C07289=1074.285,247.600,415.583,174.405,27.712,154.898
C07290=1074.292,247.848,415.555,174.407,27.716,154.899
C07291=1074.297,248.097,415.528,174.409,27.720,154.899
C07292=1074.302,248.345,415.500,174.412,27.724,154.900
C07293=1074.309,248.594,415.472,174.415,27.728,154.900
C07294=1074.318,249.000,415.427,174.419,27.734,154.901
C07295=1074.327,249.406,415.383,174.423,27.740,154.902
C07296=1074.336,249.812,415.337,174.427,27.746,154.903
C07297=1074.345,250.218,415.292,174.430,27.753,154.904
C07298=1074.351,250.466,415.265,174.433,27.757,154.905
C07299=1074.357,250.714,415.236,174.435,27.761,154.905
C07300=1074.362,250.963,415.209,174.437,27.765,154.906
C07301=1074.368,251.211,415.182,174.440,27.768,154.907
C07302=1074.374,251.459,415.153,174.442,27.772,154.907
C07303=1074.379,251.708,415.126,174.445,27.777,154.908
C07304=1074.386,251.957,415.098,174.448,27.780,154.908
C07305=1074.391,252.205,415.070,174.450,27.784,154.909
C07306=1074.397,252.453,415.042,174.452,27.788,154.910
C07307=1074.404,252.701,415.015,174.455,27.792,154.910
C07308=1074.409,252.950,414.988,174.457,27.796,154.911
C07309=1074.414,253.199,414.959,174.459,27.799,154.911
C07310=1074.421,253.446,414.932,174.462,27.803,154.912
C07311=1074.427,253.695,414.904,174.465,27.807,154.913
C07312=1074.432,253.943,414.876,174.467,27.811,154.913
C07313=1074.438,254.192,414.847,174.470,27.815,154.914
C07314=1074.444,254.440,414.821,174.472,27.819,154.914
C07315=1074.450,254.689,414.792,174.474,27.822,154.915
C07316=1074.455,254.937,414.764,174.476,27.826,154.916
C07317=1074.462,255.185,414.737,174.479,27.830,154.916
C07318=1074.467,255.433,414.709,174.482,27.834,154.917
C07319=1074.473,255.682,414.680,174.484,27.838,154.917
C07320=1074.478,255.930,414.652,174.487,27.842,154.918
C07321=1074.485,256.179,414.625,174.489,27.846,154.919
C07322=1074.491,256.427,414.596,174.492,27.849,154.919
C07323=1074.496,256.676,414.568,174.494,27.853,154.920
C07324=1074.502,256.924,414.540,174.497,27.857,154.920
C07325=1074.508,257.172,414.513,174.499,27.861,154.921
C07326=1074.514,257.421,414.484,174.502,27.865,154.922
C07327=1074.519,257.669,414.456,174.504,27.868,154.922
C07328=1074.525,257.918,414.428,174.507,27.872,154.923
C07329=1074.531,258.166,414.400,174.509,27.876,154.923
C07330=1074.537,258.414,414.372,174.512,27.880,154.924
C07331=1074.544,258.662,414.343,174.515,27.884,154.924
C07332=1074.550,258.911,414.315,174.517,27.888,154.925
C07333=1074.555,259.159,414.287,174.519,27.892,154.926
C07334=1074.562,259.407,414.259,174.522,27.895,154.926
C07335=1074.567,259.655,414.231,174.524,27.899,154.927
C07336=1074.573,259.904,414.203,174.527,27.903,154.927
C07337=1074.579,260.152,414.174,174.530,27.907,154.928
C07338=1074.584,260.400,414.146,174.532,27.910,154.929
C07339=1074.590,260.649,414.118,174.534,27.914,154.929
C07340=1074.597,260.898,414.090,174.537,27.918,154.930
C07341=1074.603,261.146,414.062,174.540,27.922,154.930
C07342=1074.609,261.394,414.033,174.542,27.926,154.931
C07343=1074.615,261.643,414.005,174.545,27.930,154.932
C07344=1074.621,261.891,413.976,174.547,27.934,154.932
C07345=1074.626,262.139,413.948,174.549,27.937,154.933
C07346=1074.636,262.543,413.902,174.554,27.944,154.934
C07347=1074.646,262.946,413.856,174.558,27.950,154.935
C07348=1074.656,263.349,413.810,174.562,27.956,154.936
C07349=1074.666,263.753,413.764,174.566,27.962,154.937
C07350=1074.672,264.002,413.735,174.569,27.966,154.937
C07351=1074.677,264.249,413.707,174.572,27.970,154.938
C07352=1074.683,264.498,413.678,174.574,27.974,154.938
C07353=1074.689,264.746,413.649,174.576,27.978,154.939
C07354=1074.695,264.994,413.621,174.579,27.981,154.939
C07355=1074.700,265.242,413.592,174.582,27.985,154.940
C07356=1074.706,265.491,413.563,174.584,27.989,154.941
C07357=1074.713,265.739,413.534,174.587,27.993,154.941
C07358=1074.718,265.987,413.506,174.589,27.997,154.942
C07359=1074.724,266.235,413.477,174.592,28.001,154.943
C07360=1074.730,266.484,413.449,174.595,28.005,154.943
C07361=1074.735,266.732,413.420,174.597,28.009,154.944
C07362=1074.741,266.980,413.391,174.600,28.013,154.944
C07363=1074.747,267.229,413.362,174.603,28.017,154.945
C07364=1074.753,267.477,413.333,174.605,28.020,154.946
C07365=1074.759,267.726,413.305,174.608,28.024,154.946
C07366=1074.765,267.973,413.276,174.610,28.028,154.947
C07367=1074.771,268.222,413.247,174.613,28.032,154.947
C07368=1074.776,268.470,413.218,174.616,28.036,154.948
C07369=1074.783,268.718,413.189,174.618,28.040,154.949
C07370=1074.789,268.967,413.160,174.620,28.044,154.949
C07371=1074.795,269.214,413.131,174.624,28.048,154.950
C07372=1074.800,269.463,413.103,174.626,28.052,154.950
C07373=1074.806,269.711,413.074,174.628,28.056,154.951
C07374=1074.812,269.959,413.044,174.631,28.059,154.952
C07375=1074.818,270.208,413.015,174.634,28.063,154.952
C07376=1074.823,270.456,412.987,174.636,28.067,154.953
C07377=1074.829,270.704,412.958,174.639,28.071,154.953
C07378=1074.835,270.952,412.928,174.641,28.075,154.954
C07379=1074.841,271.201,412.899,174.644,28.079,154.955
C07380=1074.847,271.449,412.870,174.647,28.083,154.955
C07381=1074.853,271.698,412.841,174.649,28.087,154.956
C07382=1074.859,271.946,412.812,174.651,28.091,154.957
C07383=1074.865,272.193,412.784,174.655,28.095,154.957
C07384=1074.870,272.442,412.754,174.657,28.099,154.958
C07385=1074.876,272.690,412.725,174.660,28.102,154.958
C07386=1074.883,272.938,412.696,174.663,28.107,154.959
C07387=1074.888,273.186,412.666,174.665,28.110,154.960
C07388=1074.894,273.435,412.637,174.668,28.114,154.960
C07389=1074.900,273.683,412.607,174.670,28.118,154.961
C07390=1074.906,273.931,412.578,174.673,28.122,154.961
C07391=1074.912,274.180,412.549,174.676,28.126,154.962
C07392=1074.918,274.428,412.520,174.678,28.130,154.963
C07393=1074.923,274.675,412.490,174.681,28.134,154.963
C07394=1074.929,274.924,412.461,174.684,28.138,154.964
C07395=1074.934,275.172,412.432,174.686,28.142,154.965
C07396=1074.941,275.420,412.403,174.688,28.146,154.965
C07397=1074.946,275.669,412.373,174.692,28.150,154.966
C07398=1074.956,276.076,412.325,174.696,28.156,154.967
C07399=1074.966,276.482,412.277,174.700,28.163,154.968
C07400=1074.976,276.888,412.229,174.704,28.169,154.969
C07401=1074.985,277.294,412.180,174.708,28.176,154.970
C07402=1074.991,277.543,412.151,174.712,28.180,154.971
C07403=1074.996,277.791,412.121,174.714,28.183,154.971
C07404=1075.003,278.039,412.092,174.716,28.187,154.972
C07405=1075.008,278.288,412.062,174.720,28.192,154.972
C07406=1075.014,278.535,412.032,174.722,28.196,154.973
C07407=1075.020,278.783,412.003,174.724,28.200,154.974
C07408=1075.026,279.032,411.973,174.728,28.203,154.974
C07409=1075.032,279.279,411.944,174.730,28.207,154.975
C07410=1075.038,279.528,411.914,174.733,28.211,154.975
C07411=1075.043,279.776,411.884,174.736,28.215,154.976
C07412=1075.050,280.025,411.854,174.738,28.219,154.977
C07413=1075.056,280.273,411.825,174.741,28.223,154.977
C07414=1075.061,280.521,411.795,174.744,28.227,154.978
C07415=1075.068,280.769,411.765,174.746,28.231,154.979
C07416=1075.074,281.017,411.736,174.749,28.235,154.979
C07417=1075.079,281.266,411.706,174.752,28.239,154.980
C07418=1075.085,281.514,411.676,174.754,28.243,154.980
C07419=1075.091,281.762,411.647,174.758,28.247,154.981
C07420=1075.097,282.010,411.616,174.760,28.251,154.982
C07421=1075.102,282.258,411.587,174.762,28.255,154.982
C07422=1075.108,282.506,411.556,174.766,28.260,154.983
C07423=1075.114,282.754,411.527,174.768,28.263,154.984
C07424=1075.120,283.002,411.496,174.770,28.267,154.984
C07425=1075.126,283.250,411.467,174.774,28.272,154.985
C07426=1075.132,283.498,411.437,174.776,28.275,154.986
C07427=1075.137,283.746,411.406,174.779,28.279,154.986
C07428=1075.143,283.994,411.377,174.782,28.283,154.987
C07429=1075.149,284.243,411.346,174.784,28.287,154.987
C07430=1075.155,284.491,411.317,174.788,28.291,154.988
C07431=1075.161,284.739,411.286,174.790,28.295,154.989
C07432=1075.167,284.987,411.256,174.792,28.299,154.989
C07433=1075.173,285.235,411.227,174.796,28.304,154.990
C07434=1075.179,285.483,411.196,174.798,28.308,154.991
C07435=1075.184,285.731,411.166,174.800,28.311,154.991
C07436=1075.191,285.980,411.136,174.804,28.316,154.992
C07437=1075.196,286.228,411.106,174.806,28.320,154.993
C07438=1075.202,286.476,411.075,174.809,28.324,154.993
C07439=1075.208,286.723,411.045,174.812,28.328,154.994
C07440=1075.213,286.972,411.015,174.814,28.332,154.995
C07441=1075.220,287.219,410.986,174.817,28.336,154.995
C07442=1075.226,287.468,410.955,174.820,28.339,154.996
C07443=1075.232,287.716,410.925,174.823,28.344,154.996
C07444=1075.238,287.964,410.895,174.826,28.348,154.997
C07445=1075.244,288.212,410.865,174.828,28.352,154.998
C07446=1075.250,288.460,410.834,174.831,28.356,154.998
C07447=1075.256,288.708,410.804,174.834,28.360,154.999
C07448=1075.262,288.956,410.773,174.837,28.364,155.000
C07449=1075.267,289.204,410.743,174.839,28.368,155.000
C07450=1075.277,289.621,410.692,174.844,28.375,155.001
C07451=1075.288,290.038,410.641,174.849,28.381,155.002
C07452=1075.297,290.454,410.590,174.853,28.389,155.004
C07453=1075.307,290.870,410.538,174.858,28.395,155.005
C07454=1075.313,291.118,410.507,174.861,28.400,155.005
C07455=1075.319,291.367,410.477,174.864,28.404,155.006
C07456=1075.325,291.615,410.446,174.866,28.408,155.007
C07457=1075.331,291.862,410.416,174.869,28.412,155.007
C07458=1075.337,292.110,410.386,174.872,28.416,155.008
C07459=1075.343,292.359,410.355,174.875,28.420,155.009
C07460=1075.348,292.607,410.324,174.878,28.424,155.009
C07461=1075.354,292.855,410.294,174.881,28.428,155.010
C07462=1075.360,293.103,410.263,174.883,28.432,155.011
C07463=1075.366,293.350,410.232,174.887,28.437,155.011
C07464=1075.372,293.598,410.202,174.889,28.441,155.012
C07465=1075.378,293.847,410.170,174.891,28.445,155.013
C07466=1075.384,294.095,410.140,174.895,28.449,155.013
C07467=1075.390,294.343,410.110,174.897,28.453,155.014
C07468=1075.396,294.591,410.078,174.900,28.457,155.015
C07469=1075.402,294.839,410.048,174.903,28.461,155.015
C07470=1075.407,295.087,410.017,174.906,28.465,155.016
C07471=1075.414,295.335,409.986,174.909,28.469,155.016
C07472=1075.420,295.582,409.955,174.912,28.474,155.017
C07473=1075.426,295.831,409.924,174.914,28.478,155.018
C07474=1075.431,296.079,409.893,174.918,28.482,155.019
C07475=1075.437,296.326,409.862,174.920,28.486,155.019
C07476=1075.444,296.575,409.832,174.923,28.490,155.020
C07477=1075.449,296.823,409.801,174.926,28.494,155.021
C07478=1075.455,297.070,409.770,174.929,28.498,155.021
C07479=1075.461,297.319,409.739,174.931,28.502,155.022
C07480=1075.466,297.567,409.708,174.935,28.507,155.023
C07481=1075.473,297.815,409.676,174.937,28.511,155.023
C07482=1075.478,298.063,409.646,174.940,28.515,155.024
C07483=1075.484,298.310,409.614,174.943,28.519,155.025
C07484=1075.490,298.559,409.583,174.946,28.523,155.025
C07485=1075.495,298.806,409.551,174.948,28.528,155.026
C07486=1075.501,299.054,409.521,174.952,28.532,155.027
C07487=1075.507,299.302,409.489,174.954,28.536,155.027
C07488=1075.513,299.550,409.458,174.957,28.541,155.028
C07489=1075.519,299.798,409.427,174.960,28.545,155.029
C07490=1075.524,300.046,409.395,174.963,28.549,155.029
C07491=1075.530,300.294,409.365,174.966,28.553,155.030
C07492=1075.536,300.542,409.333,174.969,28.558,155.031
C07493=1075.542,300.789,409.302,174.971,28.562,155.032
C07494=1075.548,301.038,409.270,174.975,28.566,155.032
C07495=1075.553,301.285,409.239,174.977,28.570,155.033
C07496=1075.560,301.533,409.207,174.980,28.575,155.034
C07497=1075.565,301.782,409.176,174.983,28.579,155.034
C07498=1075.572,302.029,409.145,174.986,28.583,155.035
C07499=1075.577,302.277,409.113,174.988,28.587,155.036
C07500=1075.582,302.525,409.082,174.992,28.592,155.036
C07501=1075.589,302.773,409.051,174.994,28.596,155.037
C07502=1075.594,302.988,409.023,174.996,28.600,155.038
C07503=1075.599,303.204,408.995,174.999,28.603,155.038
C07504=1075.605,303.420,408.968,175.002,28.607,155.039
C07505=1075.609,303.635,408.941,175.005,28.611,155.040
C07506=1075.615,303.851,408.913,175.007,28.614,155.040
C07507=1075.620,304.066,408.886,175.010,28.618,155.041
C07508=1075.625,304.282,408.859,175.012,28.622,155.041
C07509=1075.630,304.498,408.832,175.015,28.626,155.042
C07510=1075.636,304.746,408.800,175.018,28.630,155.043
C07511=1075.642,304.994,408.768,175.020,28.634,155.043
C07512=1075.648,305.241,408.737,175.024,28.638,155.044
C07513=1075.654,305.489,408.705,175.026,28.643,155.045
C07514=1075.659,305.737,408.673,175.029,28.647,155.046
C07515=1075.666,305.985,408.641,175.032,28.651,155.046
C07516=1075.671,306.232,408.610,175.035,28.656,155.047
C07517=1075.677,306.481,408.578,175.038,28.660,155.048
C07518=1075.684,306.728,408.546,175.041,28.664,155.048
C07519=1075.689,306.976,408.515,175.044,28.668,155.049
C07520=1075.695,307.224,408.483,175.046,28.673,155.050
C07521=1075.701,307.472,408.451,175.050,28.677,155.050
C07522=1075.707,307.720,408.420,175.052,28.681,155.051
C07523=1075.713,307.968,408.388,175.056,28.686,155.052
C07524=1075.719,308.216,408.356,175.059,28.690,155.053
C07525=1075.725,308.464,408.324,175.061,28.694,155.053
C07526=1075.731,308.711,408.292,175.065,28.699,155.054
C07527=1075.738,308.959,408.260,175.067,28.703,155.055
C07528=1075.743,309.207,408.228,175.070,28.707,155.055
C07529=1075.749,309.455,408.196,175.074,28.712,155.056
C07530=1075.756,309.703,408.165,175.076,28.716,155.057
C07531=1075.762,309.951,408.133,175.079,28.720,155.058
C07532=1075.767,310.198,408.101,175.083,28.725,155.058
C07533=1075.773,310.446,408.068,175.085,28.729,155.059
C07534=1075.779,310.694,408.036,175.088,28.733,155.060
C07535=1075.786,310.942,408.005,175.091,28.737,155.060
C07536=1075.792,311.190,407.973,175.094,28.742,155.061
C07537=1075.798,311.437,407.940,175.098,28.746,155.062
C07538=1075.804,311.685,407.908,175.100,28.751,155.063
C07539=1075.810,311.934,407.876,175.103,28.755,155.063
C07540=1075.816,312.181,407.843,175.107,28.759,155.064
C07541=1075.823,312.429,407.812,175.109,28.763,155.065
C07542=1075.828,312.677,407.780,175.112,28.768,155.065
C07543=1075.835,312.924,407.748,175.115,28.772,155.066
C07544=1075.841,313.172,407.716,175.118,28.776,155.067
C07545=1075.847,313.420,407.683,175.121,28.781,155.068
C07546=1075.853,313.668,407.651,175.124,28.785,155.068
C07547=1075.859,313.916,407.619,175.127,28.790,155.069
C07548=1075.866,314.164,407.587,175.131,28.794,155.070
C07549=1075.871,314.411,407.555,175.133,28.798,155.070
C07550=1075.877,314.659,407.522,175.136,28.803,155.071
C07551=1075.883,314.907,407.490,175.140,28.807,155.072
C07552=1075.889,315.155,407.457,175.142,28.811,155.073
C07553=1075.895,315.403,407.425,175.145,28.816,155.073
C07554=1075.901,315.650,407.393,175.149,28.821,155.074
C07555=1075.906,315.898,407.359,175.151,28.825,155.075
C07556=1075.912,316.146,407.327,175.154,28.830,155.076
C07557=1075.919,316.394,407.294,175.157,28.834,155.077
C07558=1075.924,316.611,407.266,175.160,28.838,155.077
C07559=1075.928,316.828,407.237,175.163,28.842,155.078
C07560=1075.933,317.045,407.209,175.165,28.846,155.079
C07561=1075.938,317.262,407.180,175.168,28.850,155.079
C07562=1075.944,317.480,407.151,175.171,28.854,155.080
C07563=1075.949,317.697,407.123,175.173,28.858,155.081
C07564=1075.954,317.914,407.094,175.176,28.862,155.081
C07565=1075.959,318.131,407.065,175.178,28.866,155.082
C07566=1075.965,318.379,407.033,175.182,28.871,155.083
C07567=1075.972,318.627,407.000,175.185,28.876,155.083
C07568=1075.977,318.875,406.967,175.187,28.880,155.084
C07569=1075.983,319.123,406.934,175.191,28.885,155.085
C07570=1075.989,319.371,406.901,175.194,28.889,155.086
C07571=1075.995,319.618,406.868,175.196,28.894,155.087
C07572=1076.001,319.866,406.836,175.200,28.898,155.087
C07573=1076.007,320.114,406.803,175.203,28.903,155.088
C07574=1076.013,320.362,406.770,175.205,28.907,155.089
C07575=1076.019,320.609,406.738,175.209,28.912,155.090
C07576=1076.024,320.857,406.705,175.212,28.917,155.090
C07577=1076.030,321.104,406.672,175.214,28.921,155.091
C07578=1076.036,321.352,406.638,175.218,28.926,155.092
C07579=1076.042,321.600,406.606,175.221,28.930,155.093
C07580=1076.049,321.847,406.573,175.224,28.935,155.094
C07581=1076.055,322.096,406.539,175.227,28.939,155.094
C07582=1076.061,322.344,406.507,175.230,28.944,155.095
C07583=1076.067,322.591,406.473,175.233,28.949,155.096
C07584=1076.073,322.839,406.440,175.236,28.953,155.097
C07585=1076.078,323.087,406.407,175.239,28.958,155.097
C07586=1076.085,323.335,406.374,175.243,28.963,155.098
C07587=1076.091,323.582,406.342,175.246,28.967,155.099
C07588=1076.096,323.830,406.308,175.248,28.972,155.100
C07589=1076.103,324.078,406.276,175.252,28.976,155.101
C07590=1076.109,324.325,406.242,175.255,28.981,155.101
C07591=1076.115,324.573,406.209,175.258,28.986,155.102
C07592=1076.120,324.820,406.175,175.261,28.990,155.103
C07593=1076.127,325.069,406.142,175.264,28.995,155.104
C07594=1076.133,325.317,406.109,175.267,29.000,155.105
C07595=1076.139,325.564,406.076,175.271,29.004,155.105
C07596=1076.145,325.812,406.042,175.273,29.009,155.106
C07597=1076.151,326.059,406.009,175.276,29.013,155.107
C07598=1076.157,326.307,405.976,175.280,29.018,155.108
C07599=1076.164,326.555,405.943,175.283,29.023,155.109
C07600=1076.170,326.803,405.909,175.285,29.028,155.109
C07601=1076.176,327.050,405.876,175.289,29.032,155.110
C07602=1076.182,327.298,405.843,175.292,29.037,155.111
C07603=1076.188,327.545,405.809,175.296,29.041,155.112
C07604=1076.194,327.794,405.776,175.299,29.046,155.113
C07605=1076.201,328.041,405.743,175.301,29.051,155.113
C07606=1076.206,328.289,405.709,175.305,29.056,155.114
C07607=1076.213,328.536,405.676,175.308,29.060,155.115
C07608=1076.219,328.784,405.642,175.311,29.065,155.116
C07609=1076.225,329.032,405.608,175.315,29.070,155.117
C07610=1076.231,329.279,405.575,175.317,29.074,155.117
C07611=1076.237,329.527,405.542,175.320,29.079,155.118
C07612=1076.244,329.775,405.508,175.324,29.084,155.119
C07613=1076.250,330.022,405.474,175.327,29.089,155.120
C07614=1076.255,330.236,405.446,175.330,29.092,155.121
C07615=1076.260,330.450,405.417,175.332,29.097,155.121
C07616=1076.266,330.665,405.388,175.335,29.101,155.122
C07617=1076.272,330.878,405.358,175.338,29.105,155.123
C07618=1076.277,331.092,405.329,175.340,29.109,155.123
C07619=1076.282,331.306,405.300,175.344,29.113,155.124
C07620=1076.287,331.520,405.271,175.346,29.117,155.125
C07621=1076.293,331.735,405.242,175.349,29.121,155.126
C07622=1076.299,331.982,405.208,175.352,29.126,155.126
C07623=1076.305,332.230,405.174,175.355,29.131,155.127
C07624=1076.310,332.477,405.140,175.359,29.136,155.128
C07625=1076.317,332.725,405.106,175.362,29.141,155.129
C07626=1076.323,332.973,405.072,175.364,29.146,155.130
C07627=1076.329,333.220,405.039,175.368,29.150,155.131
C07628=1076.335,333.468,405.005,175.371,29.156,155.132
C07629=1076.341,333.716,404.971,175.374,29.161,155.132
C07630=1076.347,333.963,404.937,175.378,29.165,155.133
C07631=1076.353,334.211,404.902,175.381,29.170,155.134
C07632=1076.359,334.458,404.868,175.384,29.175,155.135
C07633=1076.365,334.705,404.834,175.387,29.180,155.136
C07634=1076.371,334.954,404.801,175.390,29.185,155.137
C07635=1076.377,335.201,404.767,175.393,29.190,155.138
C07636=1076.384,335.449,404.732,175.397,29.195,155.138
C07637=1076.390,335.697,404.698,175.400,29.200,155.139
C07638=1076.395,335.944,404.664,175.404,29.205,155.140
C07639=1076.402,336.192,404.630,175.407,29.210,155.141
C07640=1076.408,336.439,404.596,175.410,29.215,155.142
C07641=1076.414,336.687,404.561,175.414,29.220,155.143
C07642=1076.420,336.934,404.527,175.416,29.225,155.144
C07643=1076.426,337.182,404.493,175.419,29.230,155.145
C07644=1076.432,337.430,404.459,175.423,29.235,155.145
C07645=1076.439,337.678,404.424,175.426,29.239,155.146
C07646=1076.445,337.925,404.390,175.429,29.244,155.147
C07647=1076.451,338.173,404.356,175.433,29.250,155.148
C07648=1076.457,338.420,404.322,175.436,29.255,155.149
C07649=1076.463,338.667,404.287,175.439,29.260,155.150
C07650=1076.470,338.915,404.252,175.443,29.265,155.151
C07651=1076.475,339.162,404.218,175.446,29.270,155.152
C07652=1076.481,339.410,404.183,175.448,29.275,155.153
C07653=1076.487,339.658,404.149,175.452,29.280,155.153
C07654=1076.494,339.905,404.114,175.455,29.285,155.154
C07655=1076.500,340.152,404.080,175.458,29.290,155.155
C07656=1076.506,340.400,404.046,175.462,29.295,155.156
C07657=1076.511,340.648,404.011,175.465,29.300,155.157
C07658=1076.518,340.895,403.976,175.468,29.305,155.158
C07659=1076.524,341.143,403.942,175.472,29.310,155.159
C07660=1076.530,341.391,403.908,175.475,29.316,155.160
C07661=1076.536,341.638,403.872,175.478,29.321,155.161
C07662=1076.542,341.886,403.838,175.482,29.326,155.162
C07663=1076.549,342.134,403.803,175.485,29.331,155.163
C07664=1076.555,342.380,403.769,175.488,29.336,155.163
C07665=1076.561,342.628,403.734,175.492,29.341,155.164
C07666=1076.567,342.876,403.698,175.495,29.347,155.165
C07667=1076.573,343.123,403.664,175.498,29.352,155.166
C07668=1076.580,343.370,403.629,175.502,29.357,155.167
C07669=1076.585,343.618,403.595,175.505,29.362,155.168
C07670=1076.591,343.829,403.564,175.508,29.367,155.169
C07671=1076.596,344.041,403.535,175.510,29.371,155.170
C07672=1076.602,344.252,403.505,175.513,29.376,155.170
C07673=1076.607,344.464,403.475,175.516,29.380,155.171
C07674=1076.612,344.675,403.446,175.519,29.384,155.172
C07675=1076.617,344.886,403.416,175.522,29.389,155.173
C07676=1076.622,345.097,403.385,175.524,29.393,155.174
C07677=1076.628,345.308,403.356,175.528,29.398,155.174
C07678=1076.634,345.556,403.320,175.531,29.403,155.175
C07679=1076.640,345.804,403.286,175.534,29.408,155.176
C07680=1076.646,346.051,403.251,175.538,29.414,155.177
C07681=1076.652,346.298,403.216,175.541,29.419,155.178
C07682=1076.658,346.547,403.181,175.544,29.424,155.179
C07683=1076.664,346.793,403.146,175.548,29.430,155.180
C07684=1076.670,347.041,403.110,175.551,29.435,155.181
C07685=1076.677,347.288,403.075,175.554,29.440,155.182
C07686=1076.683,347.536,403.039,175.558,29.445,155.183
C07687=1076.689,347.783,403.005,175.561,29.451,155.184
C07688=1076.695,348.031,402.969,175.564,29.456,155.185
C07689=1076.702,348.278,402.934,175.568,29.462,155.186
C07690=1076.708,348.526,402.899,175.571,29.467,155.187
C07691=1076.714,348.773,402.864,175.574,29.472,155.188
C07692=1076.720,349.020,402.828,175.578,29.478,155.189
C07693=1076.727,349.268,402.793,175.581,29.483,155.190
C07694=1076.733,349.515,402.757,175.584,29.488,155.191
C07695=1076.738,349.762,402.722,175.588,29.494,155.192
C07696=1076.745,350.010,402.687,175.591,29.500,155.193
C07697=1076.751,350.257,402.651,175.594,29.505,155.194
C07698=1076.758,350.505,402.616,175.599,29.510,155.195
C07699=1076.764,350.752,402.580,175.602,29.516,155.196
C07700=1076.769,350.999,402.545,175.605,29.521,155.197
C07701=1076.776,351.247,402.510,175.609,29.527,155.198
C07702=1076.782,351.495,402.474,175.612,29.532,155.199
C07703=1076.788,351.742,402.438,175.615,29.538,155.200
C07704=1076.795,351.990,402.403,175.619,29.543,155.201
C07705=1076.801,352.237,402.367,175.622,29.548,155.202
C07706=1076.807,352.484,402.331,175.625,29.554,155.203
C07707=1076.813,352.731,402.296,175.629,29.560,155.204
C07708=1076.819,352.979,402.260,175.632,29.565,155.205
C07709=1076.825,353.226,402.225,175.635,29.571,155.206
C07710=1076.831,353.474,402.189,175.640,29.576,155.207
C07711=1076.839,353.721,402.153,175.643,29.582,155.208
C07712=1076.845,353.968,402.117,175.646,29.588,155.209
C07713=1076.851,354.216,402.082,175.650,29.593,155.210
C07714=1076.857,354.463,402.045,175.653,29.599,155.211
C07715=1076.862,354.710,402.010,175.656,29.604,155.212
C07716=1076.869,354.957,401.973,175.660,29.610,155.213
C07717=1076.875,355.205,401.938,175.663,29.615,155.214
C07718=1076.882,355.452,401.902,175.666,29.621,155.215
C07719=1076.888,355.699,401.866,175.671,29.627,155.216
C07720=1076.894,355.947,401.830,175.674,29.633,155.217
C07721=1076.900,356.194,401.794,175.677,29.638,155.218
C07722=1076.906,356.442,401.758,175.681,29.644,155.219
C07723=1076.913,356.689,401.722,175.684,29.650,155.221
C07724=1076.919,356.936,401.686,175.687,29.655,155.222
C07725=1076.925,357.183,401.649,175.691,29.661,155.223
C07726=1076.931,357.396,401.619,175.694,29.666,155.224
C07727=1076.936,357.609,401.588,175.698,29.671,155.224
C07728=1076.942,357.822,401.556,175.700,29.676,155.225
C07729=1076.947,358.035,401.525,175.703,29.681,155.226
C07730=1076.952,358.248,401.495,175.706,29.686,155.227
C07731=1076.958,358.461,401.463,175.709,29.691,155.228
C07732=1076.963,358.674,401.432,175.713,29.696,155.229
C07733=1076.968,358.887,401.401,175.715,29.700,155.230
C07734=1076.975,359.135,401.364,175.718,29.707,155.231
C07735=1076.981,359.382,401.328,175.723,29.712,155.232
C07736=1076.987,359.629,401.292,175.726,29.718,155.233
C07737=1076.993,359.876,401.256,175.729,29.724,155.234
C07738=1077.000,360.123,401.219,175.733,29.730,155.236
C07739=1077.006,360.370,401.183,175.736,29.735,155.237
C07740=1077.013,360.618,401.146,175.740,29.742,155.238
C07741=1077.019,360.865,401.109,175.744,29.747,155.239
C07742=1077.025,361.113,401.074,175.747,29.753,155.240
C07743=1077.032,361.360,401.037,175.750,29.759,155.241
C07744=1077.037,361.607,401.000,175.754,29.765,155.242
C07745=1077.044,361.854,400.964,175.758,29.771,155.243
C07746=1077.050,362.101,400.927,175.761,29.777,155.244
C07747=1077.056,362.348,400.891,175.765,29.783,155.245
C07748=1077.063,362.596,400.854,175.768,29.789,155.247
C07749=1077.069,362.843,400.818,175.772,29.795,155.248
C07750=1077.076,363.090,400.781,175.776,29.801,155.249
C07751=1077.081,363.338,400.744,175.779,29.806,155.250
C07752=1077.088,363.585,400.708,175.782,29.813,155.251
C07753=1077.094,363.832,400.671,175.786,29.819,155.252
C07754=1077.101,364.079,400.634,175.790,29.825,155.253
C07755=1077.108,364.326,400.597,175.793,29.831,155.255
C07756=1077.113,364.573,400.560,175.797,29.837,155.256
C07757=1077.120,364.820,400.524,175.800,29.843,155.257
C07758=1077.126,365.067,400.487,175.804,29.849,155.258
C07759=1077.132,365.316,400.450,175.808,29.855,155.259
C07760=1077.139,365.562,400.413,175.811,29.861,155.260
C07761=1077.145,365.809,400.376,175.815,29.867,155.261
C07762=1077.151,366.056,400.339,175.819,29.873,155.263
C07763=1077.158,366.304,400.302,175.822,29.879,155.264
C07764=1077.164,366.551,400.265,175.825,29.885,155.265
C07765=1077.170,366.798,400.228,175.830,29.892,155.266
C07766=1077.177,367.044,400.191,175.833,29.898,155.267
C07767=1077.182,367.292,400.154,175.836,29.904,155.269
C07768=1077.189,367.539,400.117,175.841,29.910,155.270
C07769=1077.195,367.786,400.080,175.844,29.917,155.271
C07770=1077.201,368.033,400.043,175.847,29.923,155.272
C07771=1077.208,368.281,400.005,175.851,29.929,155.273
C07772=1077.214,368.528,399.969,175.855,29.936,155.275
C07773=1077.220,368.775,399.931,175.858,29.942,155.276
C07774=1077.227,369.022,399.893,175.862,29.948,155.277
C07775=1077.233,369.269,399.856,175.866,29.954,155.278
C07776=1077.240,369.515,399.819,175.869,29.960,155.279
C07777=1077.246,369.764,399.782,175.873,29.967,155.281
C07778=1077.252,370.010,399.745,175.877,29.973,155.282
C07779=1077.258,370.257,399.707,175.880,29.980,155.283
C07780=1077.265,370.504,399.670,175.884,29.986,155.284
C07781=1077.271,370.751,399.632,175.888,29.992,155.285
C07782=1077.282,371.143,399.573,175.894,30.003,155.287
C07783=1077.292,371.536,399.514,175.900,30.013,155.289
C07784=1077.298,371.782,399.476,175.903,30.019,155.291
C07785=1077.305,372.028,399.439,175.906,30.025,155.292
C07786=1077.311,372.275,399.402,175.911,30.032,155.293
C07787=1077.318,372.522,399.364,175.914,30.038,155.294
C07788=1077.324,372.769,399.326,175.917,30.045,155.296
C07789=1077.331,373.015,399.289,175.922,30.051,155.297
C07790=1077.337,373.262,399.251,175.925,30.058,155.298
C07791=1077.344,373.509,399.214,175.929,30.064,155.299
C07792=1077.350,373.756,399.176,175.933,30.070,155.301
C07793=1077.356,374.003,399.138,175.936,30.077,155.302
C07794=1077.362,374.250,399.100,175.940,30.084,155.303
C07795=1077.369,374.497,399.063,175.944,30.091,155.305
C07796=1077.376,374.743,399.024,175.948,30.097,155.306
C07797=1077.381,374.990,398.986,175.951,30.104,155.307
C07798=1077.388,375.238,398.948,175.955,30.110,155.308
C07799=1077.394,375.484,398.911,175.959,30.117,155.310
C07800=1077.401,375.732,398.873,175.962,30.123,155.311
C07801=1077.407,375.978,398.835,175.967,30.131,155.312
C07802=1077.414,376.226,398.797,175.970,30.137,155.314
C07803=1077.420,376.473,398.758,175.973,30.144,155.315
C07804=1077.426,376.719,398.721,175.978,30.151,155.316
C07805=1077.433,376.967,398.682,175.981,30.157,155.318
C07806=1077.439,377.213,398.645,175.985,30.164,155.319
C07807=1077.446,377.460,398.606,175.989,30.171,155.320
C07808=1077.452,377.707,398.569,175.993,30.178,155.322
C07809=1077.459,377.954,398.531,175.996,30.184,155.323
C07810=1077.465,378.201,398.492,176.001,30.191,155.324
C07811=1077.471,378.448,398.454,176.004,30.198,155.326
C07812=1077.478,378.695,398.416,176.008,30.205,155.327
C07813=1077.485,378.942,398.377,176.012,30.211,155.328
C07814=1077.491,379.189,398.339,176.016,30.219,155.330
C07815=1077.497,379.436,398.300,176.019,30.226,155.331
C07816=1077.505,379.683,398.263,176.023,30.232,155.332
C07817=1077.511,379.929,398.224,176.027,30.239,155.334
C07818=1077.517,380.176,398.186,176.030,30.246,155.335
C07819=1077.524,380.423,398.147,176.035,30.253,155.337
C07820=1077.530,380.670,398.110,176.039,30.260,155.338
C07821=1077.537,380.917,398.071,176.042,30.267,155.339
C07822=1077.544,381.163,398.032,176.047,30.274,155.341
C07823=1077.550,381.411,397.994,176.050,30.281,155.342
C07824=1077.557,381.658,397.955,176.054,30.288,155.343
C07825=1077.563,381.904,397.917,176.058,30.295,155.345
C07826=1077.570,382.151,397.878,176.062,30.302,155.346
C07827=1077.577,382.398,397.840,176.065,30.309,155.348
C07828=1077.583,382.645,397.800,176.070,30.316,155.349
C07829=1077.589,382.891,397.762,176.073,30.323,155.351
C07830=1077.595,383.139,397.724,176.077,30.331,155.352
C07831=1077.602,383.386,397.685,176.081,30.338,155.353
C07832=1077.608,383.632,397.646,176.085,30.345,155.355
C07833=1077.614,383.879,397.607,176.088,30.352,155.356
C07834=1077.621,384.126,397.568,176.093,30.359,155.358
C07835=1077.628,384.373,397.529,176.097,30.366,155.359
C07836=1077.634,384.608,397.492,176.100,30.373,155.361
C07837=1077.640,384.844,397.455,176.104,30.380,155.362
C07838=1077.646,385.079,397.418,176.108,30.387,155.363
C07839=1077.653,385.315,397.380,176.112,30.394,155.365
C07840=1077.659,385.551,397.343,176.116,30.401,155.366
C07841=1077.665,385.786,397.306,176.119,30.408,155.368
C07842=1077.671,386.022,397.268,176.123,30.415,155.369
C07843=1077.677,386.258,397.232,176.127,30.422,155.370
C07844=1077.684,386.504,397.192,176.130,30.430,155.372
C07845=1077.691,386.751,397.153,176.135,30.437,155.373
C07846=1077.698,386.997,397.115,176.139,30.444,155.375
C07847=1077.704,387.245,397.075,176.142,30.452,155.377
C07848=1077.711,387.491,397.036,176.147,30.459,155.378
C07849=1077.718,387.738,396.997,176.150,30.466,155.379
C07850=1077.724,387.985,396.957,176.154,30.474,155.381
C07851=1077.731,388.232,396.918,176.159,30.482,155.383
C07852=1077.737,388.478,396.880,176.162,30.489,155.384
C07853=1077.744,388.725,396.839,176.166,30.496,155.385
C07854=1077.751,388.972,396.801,176.171,30.504,155.387
C07855=1077.757,389.219,396.762,176.174,30.511,155.389
C07856=1077.764,389.465,396.722,176.179,30.519,155.390
C07857=1077.771,389.712,396.683,176.183,30.526,155.392
C07858=1077.777,389.958,396.643,176.187,30.534,155.393
C07859=1077.784,390.205,396.604,176.191,30.541,155.395
C07860=1077.791,390.451,396.564,176.195,30.549,155.396
C07861=1077.797,390.699,396.525,176.199,30.557,155.398
C07862=1077.804,390.945,396.485,176.203,30.565,155.399
C07863=1077.811,391.192,396.446,176.207,30.572,155.401
C07864=1077.818,391.439,396.406,176.211,30.580,155.403
C07865=1077.825,391.685,396.366,176.216,30.588,155.404
C07866=1077.831,391.932,396.327,176.219,30.595,155.406
C07867=1077.837,392.179,396.287,176.223,30.603,155.407
C07868=1077.845,392.425,396.247,176.228,30.611,155.409
C07869=1077.851,392.672,396.208,176.231,30.619,155.411
C07870=1077.857,392.919,396.168,176.235,30.627,155.412
C07871=1077.864,393.165,396.128,176.240,30.635,155.414
C07872=1077.871,393.412,396.088,176.244,30.643,155.415
C07873=1077.878,393.658,396.048,176.248,30.650,155.417
C07874=1077.884,393.905,396.009,176.252,30.658,155.419
C07875=1077.891,394.152,395.968,176.256,30.666,155.420
C07876=1077.898,394.398,395.929,176.261,30.674,155.422
C07877=1077.905,394.645,395.888,176.264,30.682,155.424
C07878=1077.911,394.892,395.848,176.268,30.690,155.425
C07879=1077.918,395.138,395.808,176.273,30.698,155.427
C07880=1077.924,395.385,395.768,176.277,30.706,155.429
C07881=1077.932,395.632,395.728,176.281,30.715,155.430
C07882=1077.938,395.878,395.688,176.285,30.723,155.432
C07883=1077.944,396.125,395.648,176.289,30.731,155.434
C07884=1077.951,396.371,395.608,176.294,30.739,155.435
C07885=1077.958,396.618,395.567,176.298,30.747,155.437
C07886=1077.965,396.865,395.528,176.302,30.755,155.439
C07887=1077.971,397.111,395.487,176.306,30.763,155.441
C07888=1077.979,397.358,395.446,176.310,30.771,155.442
C07889=1077.985,397.604,395.406,176.314,30.780,155.444
C07890=1077.991,397.851,395.366,176.319,30.788,155.446
C07891=1077.998,398.098,395.325,176.323,30.796,155.447
C07892=1078.005,398.340,395.286,176.326,30.804,155.449
C07893=1078.011,398.584,395.246,176.331,30.812,155.451
C07894=1078.018,398.826,395.206,176.335,30.820,155.452
C07895=1078.025,399.069,395.166,176.340,30.829,155.454
C07896=1078.032,399.313,395.126,176.344,30.837,155.456
C07897=1078.038,399.555,395.086,176.347,30.845,155.458
C07898=1078.045,399.799,395.046,176.352,30.854,155.460
C07899=1078.052,400.041,395.006,176.356,30.862,155.461
C07900=1078.059,400.288,394.965,176.361,30.871,155.463
C07901=1078.065,400.534,394.924,176.365,30.879,155.465
C07902=1078.072,400.781,394.884,176.369,30.888,155.467
C07903=1078.079,401.027,394.843,176.374,30.896,155.468
C07904=1078.086,401.274,394.802,176.378,30.905,155.470
C07905=1078.093,401.520,394.762,176.382,30.913,155.472
C07906=1078.099,401.767,394.720,176.386,30.922,155.474
C07907=1078.106,402.014,394.680,176.390,30.931,155.476
C07908=1078.113,402.260,394.638,176.395,30.939,155.477
C07909=1078.120,402.506,394.598,176.399,30.948,155.479
C07910=1078.127,402.753,394.557,176.403,30.957,155.481
C07911=1078.134,403.000,394.516,176.408,30.965,155.483
C07912=1078.141,403.246,394.475,176.412,30.974,155.485
C07913=1078.148,403.492,394.434,176.417,30.983,155.487
C07914=1078.154,403.740,394.393,176.421,30.992,155.489
C07915=1078.161,403.986,394.352,176.425,31.000,155.490
C07916=1078.168,404.232,394.311,176.430,31.009,155.492
C07917=1078.175,404.479,394.269,176.434,31.018,155.494
C07918=1078.181,404.725,394.228,176.439,31.027,155.496
C07919=1078.189,404.972,394.187,176.443,31.036,155.498
C07920=1078.196,405.218,394.145,176.447,31.045,155.500
C07921=1078.202,405.465,394.104,176.452,31.054,155.502
C07922=1078.209,405.711,394.063,176.456,31.063,155.504
C07923=1078.216,405.958,394.021,176.461,31.072,155.506
C07924=1078.222,406.204,393.980,176.465,31.081,155.508
C07925=1078.230,406.450,393.939,176.470,31.090,155.510
C07926=1078.237,406.697,393.898,176.474,31.099,155.512
C07927=1078.244,406.943,393.855,176.479,31.109,155.514
C07928=1078.251,407.189,393.814,176.484,31.118,155.515
C07929=1078.257,407.436,393.772,176.488,31.127,155.517
C07930=1078.264,407.683,393.731,176.493,31.136,155.519
C07931=1078.271,407.929,393.689,176.497,31.145,155.521
C07932=1078.278,408.175,393.648,176.501,31.155,155.523
C07933=1078.284,408.422,393.606,176.506,31.164,155.526
C07934=1078.292,408.668,393.564,176.510,31.173,155.527
C07935=1078.299,408.915,393.522,176.515,31.183,155.529
C07936=1078.305,409.162,393.480,176.520,31.192,155.532
C07937=1078.313,409.408,393.438,176.525,31.202,155.534
C07938=1078.319,409.654,393.397,176.529,31.211,155.536
C07939=1078.326,409.900,393.355,176.533,31.220,155.538
C07940=1078.333,410.147,393.313,176.538,31.230,155.540
C07941=1078.340,410.393,393.271,176.542,31.239,155.542
C07942=1078.347,410.639,393.229,176.548,31.249,155.544
C07943=1078.354,410.886,393.187,176.552,31.259,155.546
C07944=1078.361,411.132,393.145,176.557,31.268,155.548
C07945=1078.368,411.378,393.102,176.561,31.278,155.550
C07946=1078.376,411.625,393.061,176.566,31.287,155.552
C07947=1078.382,411.871,393.019,176.571,31.297,155.554
C07948=1078.389,412.115,392.977,176.575,31.307,155.556
C07949=1078.396,412.360,392.934,176.580,31.316,155.558
C07950=1078.404,412.603,392.893,176.584,31.326,155.560
C07951=1078.410,412.848,392.852,176.590,31.336,155.563
C07952=1078.418,413.092,392.809,176.594,31.345,155.565
C07953=1078.424,413.336,392.768,176.599,31.355,155.567
C07954=1078.431,413.580,392.726,176.603,31.364,155.569
C07955=1078.438,413.825,392.683,176.608,31.374,155.571
C07956=1078.446,414.071,392.641,176.613,31.385,155.573
C07957=1078.453,414.317,392.599,176.618,31.394,155.575
C07958=1078.460,414.563,392.556,176.622,31.404,155.578
C07959=1078.467,414.809,392.514,176.628,31.414,155.580
C07960=1078.474,415.055,392.471,176.632,31.424,155.582
C07961=1078.482,415.302,392.428,176.638,31.434,155.584
C07962=1078.489,415.548,392.386,176.642,31.444,155.586
C07963=1078.496,415.795,392.343,176.647,31.454,155.589
C07964=1078.502,416.041,392.301,176.652,31.464,155.591
C07965=1078.510,416.286,392.258,176.657,31.475,155.593
C07966=1078.518,416.533,392.215,176.661,31.485,155.595
C07967=1078.525,416.779,392.172,176.667,31.495,155.598
C07968=1078.532,417.025,392.129,176.671,31.506,155.600
C07969=1078.539,417.271,392.087,176.677,31.516,155.602
C07970=1078.545,417.518,392.044,176.681,31.526,155.604
C07971=1078.553,417.764,392.001,176.687,31.537,155.607
C07972=1078.560,418.010,391.958,176.691,31.547,155.609
C07973=1078.567,418.256,391.915,176.696,31.557,155.611
C07974=1078.574,418.502,391.872,176.701,31.568,155.614
C07975=1078.581,418.749,391.828,176.706,31.578,155.616
C07976=1078.588,418.995,391.785,176.711,31.589,155.618
C07977=1078.595,419.241,391.742,176.716,31.599,155.621
C07978=1078.603,419.487,391.699,176.721,31.610,155.623
C07979=1078.610,419.734,391.656,176.726,31.621,155.625
C07980=1078.617,419.979,391.613,176.731,31.631,155.628
C07981=1078.625,420.226,391.569,176.736,31.642,155.630
C07982=1078.632,420.471,391.526,176.741,31.653,155.632
C07983=1078.640,420.718,391.482,176.747,31.664,155.635
C07984=1078.646,420.964,391.440,176.751,31.674,155.637
C07985=1078.654,421.210,391.396,176.757,31.685,155.640
C07986=1078.661,421.456,391.353,176.761,31.696,155.642
C07987=1078.669,421.702,391.309,176.767,31.707,155.645
C07988=1078.676,421.948,391.265,176.772,31.718,155.647
C07989=1078.683,422.194,391.222,176.777,31.729,155.649
C07990=1078.690,422.440,391.179,176.783,31.740,155.652
C07991=1078.697,422.686,391.135,176.787,31.751,155.654
C07992=1078.705,422.933,391.091,176.793,31.762,155.657
C07993=1078.712,423.178,391.048,176.798,31.773,155.659
C07994=1078.719,423.424,391.003,176.803,31.784,155.662
C07995=1078.726,423.670,390.960,176.809,31.795,155.664
C07996=1078.734,423.916,390.916,176.814,31.806,155.667
C07997=1078.741,424.162,390.872,176.819,31.818,155.669
C07998=1078.749,424.408,390.828,176.824,31.829,155.672
C07999=1078.756,424.654,390.784,176.830,31.840,155.674
C08000=1078.763,424.900,390.740,176.835,31.851,155.677
C08001=1078.771,425.146,390.696,176.840,31.863,155.680
C08002=1078.777,425.392,390.652,176.846,31.874,155.682
C08003=1078.785,425.638,390.608,176.851,31.886,155.685
C08004=1078.793,425.897,390.561,176.857,31.898,155.687
C08005=1078.801,426.156,390.515,176.863,31.910,155.690
C08006=1078.809,426.416,390.468,176.868,31.922,155.693
C08007=1078.817,426.675,390.422,176.874,31.934,155.696
C08008=1078.825,426.921,390.377,176.879,31.946,155.698
C08009=1078.831,427.167,390.334,176.884,31.957,155.701
C08010=1078.839,427.412,390.289,176.890,31.969,155.704
C08011=1078.846,427.658,390.244,176.895,31.981,155.706
C08012=1078.855,427.904,390.200,176.901,31.993,155.709
C08013=1078.862,428.151,390.156,176.907,32.005,155.712
C08014=1078.869,428.396,390.112,176.912,32.017,155.714
C08015=1078.876,428.642,390.067,176.917,32.028,155.717
C08016=1078.884,428.888,390.022,176.923,32.040,155.720
C08017=1078.892,429.134,389.978,176.928,32.052,155.722
C08018=1078.898,429.379,389.933,176.934,32.064,155.725
C08019=1078.906,429.625,389.888,176.940,32.076,155.728
C08020=1078.914,429.871,389.844,176.945,32.088,155.731
C08021=1078.921,430.117,389.799,176.951,32.101,155.734
C08022=1078.929,430.363,389.754,176.957,32.113,155.736
C08023=1078.937,430.609,389.710,176.962,32.125,155.739
C08024=1078.944,430.854,389.664,176.968,32.137,155.742
C08025=1078.952,431.100,389.619,176.974,32.150,155.745
C08026=1078.959,431.346,389.574,176.980,32.162,155.748
C08027=1078.967,431.592,389.530,176.985,32.174,155.750
C08028=1078.975,431.837,389.484,176.991,32.187,155.753
C08029=1078.982,432.083,389.439,176.997,32.199,155.756
C08030=1078.990,432.329,389.393,177.003,32.211,155.759
C08031=1078.997,432.575,389.349,177.008,32.224,155.762
C08032=1079.005,432.820,389.303,177.014,32.237,155.765
C08033=1079.012,433.066,389.258,177.020,32.249,155.768
C08034=1079.020,433.312,389.213,177.026,32.262,155.771
C08035=1079.028,433.558,389.168,177.031,32.275,155.774
C08036=1079.035,433.803,389.122,177.037,32.287,155.777
C08037=1079.043,434.048,389.077,177.043,32.300,155.779
C08038=1079.050,434.295,389.032,177.049,32.313,155.782
C08039=1079.058,434.540,388.986,177.054,32.326,155.785
C08040=1079.066,434.785,388.940,177.060,32.339,155.788
C08041=1079.073,435.031,388.895,177.066,32.352,155.791
C08042=1079.081,435.276,388.849,177.072,32.365,155.794
C08043=1079.088,435.522,388.804,177.079,32.378,155.797
C08044=1079.096,435.768,388.758,177.085,32.391,155.801
C08045=1079.104,436.014,388.713,177.090,32.404,155.804
C08046=1079.111,436.260,388.666,177.096,32.417,155.807
C08047=1079.119,436.505,388.621,177.102,32.430,155.810
C08048=1079.126,436.750,388.574,177.109,32.444,155.813
C08049=1079.135,436.996,388.528,177.115,32.457,155.816
C08050=1079.142,437.241,388.483,177.121,32.470,155.819
C08051=1079.150,437.487,388.437,177.126,32.484,155.822
C08052=1079.158,437.733,388.391,177.133,32.497,155.825
C08053=1079.166,437.978,388.345,177.139,32.511,155.829
C08054=1079.174,438.223,388.299,177.145,32.524,155.832
C08055=1079.182,438.469,388.253,177.151,32.538,155.835
C08056=1079.190,438.715,388.207,177.158,32.551,155.838
C08057=1079.198,438.960,388.161,177.164,32.565,155.841
C08058=1079.205,439.206,388.114,177.170,32.578,155.844
C08059=1079.214,439.452,388.068,177.177,32.592,155.848
C08060=1079.226,439.851,387.992,177.187,32.615,155.853
C08061=1079.239,440.251,387.917,177.197,32.637,155.858
C08062=1079.252,440.651,387.841,177.207,32.660,155.864
C08063=1079.265,441.051,387.765,177.217,32.683,155.869
C08064=1079.272,441.296,387.719,177.224,32.697,155.873
C08065=1079.281,441.542,387.672,177.230,32.712,155.876
C08066=1079.288,441.787,387.626,177.237,32.726,155.879
C08067=1079.296,442.033,387.578,177.243,32.740,155.883
C08068=1079.305,442.278,387.531,177.250,32.754,155.886
C08069=1079.312,442.523,387.485,177.256,32.768,155.889
C08070=1079.321,442.769,387.438,177.263,32.783,155.893
C08071=1079.328,443.014,387.391,177.270,32.797,155.896
C08072=1079.336,443.259,387.344,177.277,32.812,155.900
C08073=1079.344,443.505,387.296,177.283,32.827,155.903
C08074=1079.352,443.749,387.250,177.290,32.842,155.907
C08075=1079.360,443.995,387.202,177.296,32.856,155.910
C08076=1079.369,444.241,387.156,177.303,32.871,155.914
C08077=1079.377,444.486,387.108,177.309,32.885,155.917
C08078=1079.385,444.731,387.061,177.316,32.900,155.921
C08079=1079.393,444.977,387.014,177.323,32.915,155.924
C08080=1079.401,445.222,386.966,177.329,32.930,155.928
C08081=1079.409,445.467,386.919,177.336,32.945,155.932
C08082=1079.417,445.712,386.871,177.344,32.960,155.935
C08083=1079.425,445.958,386.824,177.350,32.975,155.939
C08084=1079.433,446.202,386.777,177.357,32.991,155.943
C08085=1079.442,446.448,386.729,177.363,33.006,155.946
C08086=1079.450,446.693,386.681,177.369,33.021,155.950
C08087=1079.458,446.938,386.634,177.376,33.036,155.954
C08088=1079.466,447.184,386.586,177.381,33.051,155.957
C08089=1079.474,447.429,386.538,177.386,33.066,155.961
C08090=1079.483,447.674,386.490,177.391,33.081,155.965
C08091=1079.491,447.919,386.442,177.397,33.096,155.968
C08092=1079.500,448.164,386.394,177.402,33.111,155.972
C08093=1079.508,448.409,386.346,177.406,33.127,155.976
C08094=1079.516,448.655,386.298,177.410,33.141,155.980
C08095=1079.525,448.899,386.251,177.415,33.157,155.983
C08096=1079.533,449.144,386.204,177.418,33.171,155.987
C08097=1079.543,449.389,386.156,177.422,33.186,155.991
C08098=1079.555,449.635,386.111,177.426,33.199,155.994
C08099=1079.568,449.880,386.066,177.429,33.211,155.997
C08100=1079.204,449.874,385.841,177.404,33.377,156.041
C08101=1079.191,449.629,385.886,177.401,33.364,156.038
C08102=1079.179,449.383,385.931,177.396,33.351,156.034
C08103=1079.168,449.138,385.978,177.393,33.337,156.031
C08104=1079.159,448.893,386.026,177.389,33.322,156.027
C08105=1079.151,448.648,386.074,177.384,33.307,156.023
C08106=1079.143,448.403,386.122,177.380,33.292,156.020
C08107=1079.134,448.158,386.170,177.375,33.277,156.016
C08108=1079.126,447.913,386.218,177.371,33.262,156.012
C08109=1079.118,447.668,386.266,177.366,33.246,156.008
C08110=1079.110,447.422,386.314,177.360,33.231,156.005
C08111=1079.101,447.178,386.361,177.355,33.217,156.001
C08112=1079.093,446.932,386.409,177.349,33.201,155.997
C08113=1079.084,446.687,386.457,177.342,33.186,155.994
C08114=1079.077,446.441,386.505,177.336,33.171,155.990
C08115=1079.068,446.196,386.552,177.330,33.156,155.986
C08116=1079.060,445.951,386.600,177.323,33.141,155.983
C08117=1079.052,445.705,386.647,177.316,33.126,155.979
C08118=1079.044,445.461,386.695,177.309,33.110,155.975
C08119=1079.036,445.216,386.743,177.302,33.095,155.972
C08120=1079.028,444.970,386.790,177.296,33.080,155.968
C08121=1079.019,444.725,386.837,177.288,33.066,155.965
C08122=1079.011,444.479,386.885,177.281,33.051,155.961
C08123=1079.004,444.235,386.932,177.275,33.036,155.957
C08124=1078.995,443.989,386.979,177.268,33.021,155.954
C08125=1078.987,443.744,387.026,177.262,33.006,155.950
C08126=1078.978,443.499,387.074,177.254,32.992,155.947
C08127=1078.971,443.254,387.121,177.247,32.977,155.943
C08128=1078.963,443.008,387.167,177.241,32.963,155.940
C08129=1078.955,442.762,387.215,177.234,32.948,155.936
C08130=1078.947,442.517,387.261,177.228,32.934,155.933
C08131=1078.939,442.272,387.309,177.221,32.920,155.930
C08132=1078.930,442.027,387.356,177.215,32.905,155.926
C08133=1078.923,441.781,387.402,177.207,32.891,155.923
C08134=1078.915,441.536,387.449,177.201,32.877,155.919
C08135=1078.907,441.291,387.495,177.195,32.862,155.916
C08136=1078.899,441.045,387.543,177.188,32.848,155.913
C08137=1078.886,440.662,387.616,177.178,32.827,155.907
C08138=1078.874,440.278,387.688,177.168,32.804,155.902
C08139=1078.862,439.896,387.761,177.158,32.783,155.897
C08140=1078.849,439.513,387.833,177.148,32.761,155.892
C08141=1078.842,439.267,387.879,177.142,32.747,155.889
C08142=1078.833,439.022,387.926,177.136,32.734,155.885
C08143=1078.825,438.776,387.972,177.129,32.720,155.882
C08144=1078.818,438.531,388.019,177.123,32.707,155.879
C08145=1078.810,438.285,388.064,177.117,32.693,155.876
C08146=1078.801,438.040,388.111,177.110,32.680,155.873
C08147=1078.794,437.794,388.157,177.104,32.666,155.870
C08148=1078.786,437.549,388.203,177.098,32.653,155.866
C08149=1078.778,437.303,388.249,177.092,32.639,155.863
C08150=1078.770,437.058,388.295,177.085,32.626,155.860
C08151=1078.762,436.812,388.341,177.079,32.613,155.857
C08152=1078.754,436.566,388.387,177.073,32.599,155.854
C08153=1078.746,436.321,388.432,177.067,32.586,155.851
C08154=1078.739,436.075,388.478,177.061,32.573,155.848
C08155=1078.731,435.830,388.523,177.054,32.559,155.845
C08156=1078.723,435.584,388.570,177.048,32.547,155.842
C08157=1078.716,435.338,388.616,177.043,32.533,155.839
C08158=1078.708,435.093,388.661,177.037,32.521,155.836
C08159=1078.701,434.847,388.707,177.031,32.508,155.833
C08160=1078.693,434.602,388.753,177.025,32.495,155.829
C08161=1078.685,434.356,388.798,177.019,32.482,155.826
C08162=1078.677,434.110,388.844,177.013,32.469,155.824
C08163=1078.670,433.865,388.890,177.006,32.456,155.821
C08164=1078.662,433.619,388.935,177.000,32.443,155.818
C08165=1078.654,433.374,388.980,176.995,32.430,155.815
C08166=1078.646,433.128,389.026,176.989,32.418,155.812
C08167=1078.639,432.882,389.071,176.983,32.405,155.809
C08168=1078.631,432.637,389.116,176.977,32.392,155.806
C08169=1078.624,432.391,389.161,176.971,32.380,155.803
C08170=1078.616,432.145,389.207,176.965,32.367,155.800
C08171=1078.609,431.899,389.252,176.960,32.355,155.797
C08172=1078.601,431.654,389.297,176.954,32.343,155.794
C08173=1078.594,431.408,389.342,176.948,32.330,155.791
C08174=1078.586,431.162,389.387,176.942,32.318,155.789
C08175=1078.578,430.916,389.432,176.936,32.306,155.786
C08176=1078.571,430.670,389.477,176.931,32.294,155.783
C08177=1078.563,430.425,389.522,176.925,32.281,155.780
C08178=1078.556,430.179,389.566,176.919,32.269,155.777
C08179=1078.548,429.933,389.612,176.914,32.257,155.775
C08180=1078.540,429.687,389.656,176.908,32.245,155.772
C08181=1078.533,429.441,389.701,176.903,32.233,155.769
C08182=1078.526,429.196,389.746,176.897,32.221,155.766
C08183=1078.518,428.950,389.791,176.891,32.209,155.764
C08184=1078.510,428.704,389.835,176.885,32.197,155.761
C08185=1078.503,428.458,389.880,176.880,32.185,155.758
C08186=1078.496,428.212,389.925,176.874,32.173,155.755
C08187=1078.488,427.966,389.969,176.869,32.161,155.753
C08188=1078.481,427.721,390.014,176.863,32.149,155.750
C08189=1078.473,427.475,390.058,176.858,32.137,155.747
C08190=1078.466,427.229,390.103,176.852,32.126,155.745
C08191=1078.458,426.983,390.147,176.846,32.114,155.742
C08192=1078.450,426.737,390.191,176.842,32.103,155.739
C08193=1078.443,426.476,390.238,176.835,32.090,155.737
C08194=1078.435,426.216,390.284,176.829,32.078,155.734
C08195=1078.426,425.955,390.332,176.824,32.066,155.731
C08196=1078.419,425.694,390.378,176.818,32.054,155.728
C08197=1078.411,425.449,390.423,176.812,32.042,155.726
C08198=1078.404,425.202,390.467,176.808,32.031,155.723
C08199=1078.397,424.957,390.511,176.802,32.020,155.721
C08200=1078.389,424.711,390.555,176.796,32.008,155.718
C08201=1078.382,424.465,390.599,176.791,31.997,155.715
C08202=1078.374,424.219,390.643,176.786,31.985,155.713
C08203=1078.367,423.973,390.686,176.780,31.975,155.710
C08204=1078.360,423.727,390.731,176.775,31.963,155.708
C08205=1078.352,423.481,390.774,176.770,31.952,155.705
C08206=1078.346,423.235,390.818,176.764,31.941,155.703
C08207=1078.338,422.988,390.862,176.760,31.929,155.700
C08208=1078.330,422.743,390.906,176.754,31.918,155.698
C08209=1078.323,422.497,390.950,176.748,31.907,155.695
C08210=1078.316,422.251,390.993,176.744,31.897,155.693
C08211=1078.309,422.005,391.037,176.738,31.885,155.690
C08212=1078.301,421.759,391.080,176.733,31.874,155.688
C08213=1078.294,421.512,391.125,176.728,31.864,155.685
C08214=1078.287,421.267,391.168,176.722,31.853,155.683
C08215=1078.279,421.020,391.211,176.718,31.842,155.681
C08216=1078.272,420.775,391.255,176.712,31.831,155.678
C08217=1078.264,420.528,391.298,176.707,31.821,155.676
C08218=1078.258,420.282,391.341,176.702,31.810,155.673
C08219=1078.250,420.036,391.384,176.697,31.799,155.671
C08220=1078.243,419.790,391.428,176.691,31.788,155.669
C08221=1078.236,419.544,391.471,176.687,31.778,155.666
C08222=1078.228,419.298,391.515,176.681,31.767,155.664
C08223=1078.221,419.052,391.557,176.677,31.757,155.662
C08224=1078.214,418.805,391.601,176.671,31.746,155.659
C08225=1078.207,418.559,391.645,176.666,31.736,155.657
C08226=1078.200,418.313,391.687,176.661,31.725,155.655
C08227=1078.192,418.067,391.731,176.656,31.715,155.652
C08228=1078.185,417.820,391.773,176.651,31.704,155.650
C08229=1078.178,417.575,391.817,176.646,31.694,155.648
C08230=1078.171,417.328,391.859,176.642,31.683,155.645
C08231=1078.163,417.082,391.903,176.636,31.673,155.643
C08232=1078.157,416.836,391.945,176.631,31.663,155.641
C08233=1078.150,416.590,391.988,176.626,31.652,155.638
C08234=1078.143,416.344,392.031,176.621,31.642,155.636
C08235=1078.136,416.098,392.074,176.617,31.632,155.634
C08236=1078.128,415.851,392.116,176.611,31.622,155.632
C08237=1078.121,415.605,392.160,176.607,31.612,155.629
C08238=1078.114,415.359,392.202,176.601,31.602,155.627
C08239=1078.107,415.113,392.244,176.597,31.592,155.625
C08240=1078.099,414.866,392.287,176.592,31.582,155.623
C08241=1078.092,414.619,392.330,176.587,31.572,155.621
C08242=1078.085,414.373,392.372,176.582,31.562,155.619
C08243=1078.078,414.128,392.415,176.577,31.552,155.616
C08244=1078.071,413.881,392.457,176.572,31.542,155.614
C08245=1078.064,413.636,392.499,176.567,31.532,155.612
C08246=1078.056,413.392,392.541,176.563,31.522,155.610
C08247=1078.049,413.147,392.584,176.558,31.512,155.608
C08248=1078.042,412.902,392.625,176.553,31.503,155.606
C08249=1078.035,412.657,392.667,176.548,31.493,155.603
C08250=1078.028,412.412,392.710,176.544,31.483,155.601
C08251=1078.021,412.167,392.751,176.539,31.474,155.599
C08252=1078.013,411.923,392.794,176.535,31.464,155.597
C08253=1078.007,411.676,392.835,176.529,31.454,155.595
C08254=1078.000,411.429,392.878,176.525,31.445,155.593
C08255=1077.992,411.183,392.920,176.520,31.435,155.591
C08256=1077.985,410.937,392.962,176.516,31.426,155.589
C08257=1077.979,410.690,393.004,176.510,31.416,155.587
C08258=1077.971,410.444,393.046,176.506,31.406,155.585
C08259=1077.964,410.198,393.089,176.501,31.397,155.583
C08260=1077.957,409.951,393.130,176.497,31.387,155.580
C08261=1077.951,409.706,393.172,176.492,31.378,155.578
C08262=1077.944,409.459,393.214,176.488,31.368,155.576
C08263=1077.937,409.213,393.256,176.482,31.359,155.574
C08264=1077.930,408.966,393.298,176.478,31.350,155.572
C08265=1077.923,408.720,393.340,176.473,31.340,155.570
C08266=1077.916,408.473,393.381,176.469,31.331,155.568
C08267=1077.908,408.227,393.423,176.464,31.322,155.566
C08268=1077.902,407.981,393.465,176.460,31.312,155.564
C08269=1077.895,407.734,393.506,176.455,31.303,155.562
C08270=1077.888,407.488,393.549,176.451,31.294,155.560
C08271=1077.881,407.241,393.590,176.446,31.284,155.558
C08272=1077.874,406.995,393.632,176.442,31.275,155.556
C08273=1077.868,406.749,393.673,176.437,31.266,155.554
C08274=1077.861,406.502,393.715,176.432,31.257,155.552
C08275=1077.854,406.256,393.756,176.427,31.248,155.550
C08276=1077.846,406.009,393.798,176.423,31.239,155.548
C08277=1077.840,405.763,393.839,176.419,31.230,155.547
C08278=1077.833,405.516,393.880,176.414,31.221,155.545
C08279=1077.827,405.269,393.922,176.410,31.212,155.543
C08280=1077.819,405.023,393.963,176.405,31.203,155.541
C08281=1077.813,404.777,394.004,176.401,31.194,155.539
C08282=1077.805,404.530,394.045,176.396,31.185,155.537
C08283=1077.799,404.283,394.087,176.392,31.176,155.535
C08284=1077.792,404.038,394.128,176.387,31.167,155.533
C08285=1077.785,403.791,394.169,176.383,31.158,155.531
C08286=1077.778,403.544,394.211,176.378,31.150,155.529
C08287=1077.772,403.298,394.252,176.374,31.141,155.528
C08288=1077.765,403.051,394.293,176.369,31.132,155.526
C08289=1077.757,402.804,394.334,176.365,31.123,155.524
C08290=1077.751,402.558,394.375,176.361,31.115,155.522
C08291=1077.743,402.312,394.416,176.357,31.106,155.520
C08292=1077.736,402.065,394.457,176.353,31.097,155.518
C08293=1077.730,401.819,394.497,176.348,31.089,155.516
C08294=1077.722,401.572,394.538,176.344,31.080,155.515
C08295=1077.716,401.326,394.580,176.339,31.071,155.513
C08296=1077.709,401.079,394.620,176.335,31.063,155.511
C08297=1077.703,400.833,394.661,176.331,31.054,155.509
C08298=1077.696,400.586,394.702,176.326,31.046,155.507
C08299=1077.689,400.340,394.743,176.322,31.037,155.506
C08300=1077.682,400.093,394.783,176.317,31.029,155.504
C08301=1077.676,399.849,394.823,176.314,31.020,155.502
C08302=1077.669,399.605,394.864,176.309,31.012,155.500
C08303=1077.662,399.362,394.904,176.305,31.004,155.498
C08304=1077.655,399.119,394.944,176.300,30.995,155.497
C08305=1077.649,398.875,394.984,176.296,30.987,155.495
C08306=1077.642,398.632,395.024,176.293,30.979,155.493
C08307=1077.635,398.387,395.065,176.288,30.971,155.492
C08308=1077.628,398.144,395.105,176.284,30.963,155.490
C08309=1077.621,397.898,395.145,176.279,30.954,155.488
C08310=1077.614,397.651,395.185,176.275,30.946,155.486
C08311=1077.608,397.404,395.225,176.271,30.938,155.485
C08312=1077.601,397.158,395.266,176.267,30.929,155.483
C08313=1077.594,396.911,395.307,176.263,30.921,155.481
C08314=1077.588,396.664,395.347,176.258,30.913,155.479
C08315=1077.581,396.418,395.386,176.254,30.905,155.478
C08316=1077.574,396.171,395.427,176.250,30.897,155.476
C08317=1077.567,395.924,395.467,176.246,30.888,155.474
C08318=1077.561,395.678,395.507,176.242,30.880,155.473
C08319=1077.554,395.431,395.548,176.237,30.872,155.471
C08320=1077.548,395.184,395.588,176.233,30.864,155.469
C08321=1077.541,394.938,395.627,176.229,30.856,155.468
C08322=1077.534,394.692,395.667,176.225,30.848,155.466
C08323=1077.528,394.445,395.708,176.220,30.840,155.464
C08324=1077.521,394.198,395.748,176.216,30.832,155.463
C08325=1077.514,393.952,395.788,176.213,30.824,155.461
C08326=1077.507,393.705,395.828,176.208,30.817,155.459
C08327=1077.501,393.459,395.868,176.204,30.809,155.458
C08328=1077.493,393.212,395.908,176.199,30.800,155.456
C08329=1077.487,392.965,395.948,176.196,30.793,155.454
C08330=1077.480,392.718,395.987,176.192,30.785,155.453
C08331=1077.474,392.472,396.027,176.187,30.777,155.451
C08332=1077.467,392.225,396.067,176.184,30.769,155.450
C08333=1077.460,391.979,396.107,176.179,30.761,155.448
C08334=1077.454,391.731,396.146,176.175,30.754,155.446
C08335=1077.447,391.485,396.187,176.171,30.746,155.445
C08336=1077.440,391.239,396.226,176.167,30.738,155.443
C08337=1077.433,390.992,396.265,176.163,30.731,155.442
C08338=1077.427,390.745,396.305,176.158,30.723,155.440
C08339=1077.420,390.498,396.344,176.155,30.715,155.438
C08340=1077.414,390.252,396.384,176.151,30.708,155.437
C08341=1077.407,390.005,396.423,176.146,30.700,155.435
C08342=1077.400,389.759,396.463,176.143,30.693,155.434
C08343=1077.394,389.512,396.502,176.138,30.685,155.432
C08344=1077.386,389.266,396.542,176.134,30.677,155.431
C08345=1077.379,389.018,396.581,176.131,30.670,155.429
C08346=1077.373,388.771,396.621,176.126,30.662,155.428
C08347=1077.366,388.525,396.660,176.122,30.655,155.426
C08348=1077.360,388.277,396.699,176.118,30.647,155.425
C08349=1077.353,388.031,396.739,176.114,30.640,155.423
C08350=1077.346,387.784,396.778,176.110,30.632,155.422
C08351=1077.340,387.537,396.817,176.106,30.625,155.420
C08352=1077.333,387.292,396.856,176.102,30.618,155.419
C08353=1077.326,387.045,396.895,176.098,30.610,155.417
C08354=1077.320,386.798,396.934,176.094,30.602,155.416
C08355=1077.314,386.551,396.973,176.090,30.595,155.414
C08356=1077.307,386.304,397.012,176.086,30.588,155.413
C08357=1077.300,386.068,397.050,176.082,30.581,155.411
C08358=1077.294,385.831,397.088,176.079,30.574,155.410
C08359=1077.288,385.596,397.125,176.074,30.567,155.408
C08360=1077.281,385.359,397.162,176.071,30.560,155.407
C08361=1077.275,385.122,397.199,176.067,30.553,155.405
C08362=1077.269,384.887,397.237,176.063,30.546,155.404
C08363=1077.262,384.650,397.274,176.059,30.539,155.403
C08364=1077.256,384.415,397.311,176.056,30.532,155.401
C08365=1077.250,384.168,397.351,176.052,30.525,155.400
C08366=1077.243,383.921,397.390,176.047,30.517,155.398
C08367=1077.237,383.673,397.428,176.044,30.510,155.397
C08368=1077.230,383.427,397.466,176.040,30.503,155.395
C08369=1077.224,383.180,397.506,176.036,30.496,155.394
C08370=1077.217,382.933,397.544,176.032,30.488,155.392
C08371=1077.211,382.686,397.583,176.028,30.482,155.391
C08372=1077.204,382.440,397.622,176.024,30.474,155.390
C08373=1077.198,382.193,397.661,176.021,30.467,155.388
C08374=1077.192,381.946,397.699,176.016,30.460,155.387
C08375=1077.185,381.699,397.738,176.013,30.453,155.385
C08376=1077.179,381.453,397.777,176.009,30.446,155.384
C08377=1077.172,381.205,397.815,176.005,30.439,155.383
C08378=1077.166,380.958,397.854,176.001,30.432,155.381
C08379=1077.159,380.712,397.892,175.997,30.425,155.380
C08380=1077.153,380.465,397.930,175.993,30.418,155.378
C08381=1077.146,380.218,397.969,175.990,30.412,155.377
C08382=1077.139,379.971,398.006,175.985,30.404,155.376
C08383=1077.132,379.724,398.045,175.982,30.397,155.374
C08384=1077.126,379.478,398.084,175.978,30.391,155.373
C08385=1077.119,379.231,398.122,175.974,30.384,155.372
C08386=1077.112,378.984,398.161,175.970,30.377,155.370
C08387=1077.107,378.737,398.198,175.966,30.370,155.369
C08388=1077.100,378.490,398.237,175.962,30.363,155.367
C08389=1077.093,378.243,398.275,175.959,30.357,155.366
C08390=1077.087,377.996,398.313,175.954,30.349,155.365
C08391=1077.080,377.749,398.352,175.951,30.343,155.363
C08392=1077.074,377.502,398.390,175.947,30.336,155.362
C08393=1077.067,377.255,398.427,175.943,30.329,155.361
C08394=1077.061,377.008,398.466,175.940,30.323,155.359
C08395=1077.055,376.762,398.504,175.935,30.316,155.358
C08396=1077.048,376.514,398.542,175.932,30.309,155.357
C08397=1077.042,376.267,398.580,175.928,30.302,155.356
C08398=1077.035,376.021,398.619,175.924,30.296,155.354
C08399=1077.029,375.773,398.657,175.921,30.289,155.353
C08400=1077.022,375.527,398.694,175.917,30.282,155.352
C08401=1077.016,375.279,398.732,175.913,30.275,155.350
C08402=1077.010,375.033,398.770,175.909,30.269,155.349
C08403=1077.003,374.785,398.808,175.905,30.262,155.348
C08404=1076.997,374.538,398.846,175.902,30.256,155.346
C08405=1076.991,374.292,398.884,175.898,30.249,155.345
C08406=1076.984,374.045,398.922,175.894,30.243,155.344
C08407=1076.977,373.798,398.960,175.890,30.236,155.342
C08408=1076.972,373.551,398.998,175.887,30.229,155.341
C08409=1076.965,373.304,399.036,175.883,30.223,155.340
C08410=1076.959,373.057,399.072,175.879,30.216,155.339
C08411=1076.952,372.809,399.110,175.876,30.210,155.337
C08412=1076.946,372.563,399.147,175.872,30.203,155.336
C08413=1076.940,372.341,399.182,175.869,30.198,155.335
C08414=1076.934,372.119,399.216,175.865,30.192,155.334
C08415=1076.928,371.896,399.249,175.862,30.186,155.333
C08416=1076.922,371.675,399.282,175.858,30.180,155.332
C08417=1076.916,371.454,399.316,175.855,30.174,155.330
C08418=1076.910,371.232,399.351,175.852,30.168,155.329
C08419=1076.905,371.010,399.384,175.848,30.163,155.328
C08420=1076.899,370.788,399.418,175.845,30.157,155.327
C08421=1076.893,370.541,399.455,175.841,30.151,155.326
C08422=1076.887,370.293,399.492,175.838,30.144,155.325
C08423=1076.880,370.047,399.529,175.834,30.138,155.323
C08424=1076.874,369.800,399.567,175.830,30.132,155.322
C08425=1076.867,369.552,399.604,175.827,30.126,155.321
C08426=1076.861,369.306,399.642,175.823,30.119,155.320
C08427=1076.854,369.059,399.679,175.819,30.113,155.319
C08428=1076.848,368.811,399.716,175.816,30.107,155.317
C08429=1076.842,368.565,399.754,175.811,30.100,155.316
C08430=1076.835,368.317,399.791,175.808,30.094,155.315
C08431=1076.829,368.070,399.828,175.805,30.088,155.314
C08432=1076.822,367.823,399.865,175.801,30.081,155.312
C08433=1076.816,367.576,399.903,175.797,30.075,155.311
C08434=1076.810,367.329,399.939,175.794,30.069,155.310
C08435=1076.804,367.082,399.977,175.790,30.063,155.309
C08436=1076.797,366.835,400.013,175.786,30.056,155.308
C08437=1076.791,366.587,400.051,175.783,30.050,155.306
C08438=1076.785,366.340,400.088,175.779,30.044,155.305
C08439=1076.779,366.093,400.125,175.776,30.038,155.304
C08440=1076.772,365.847,400.162,175.771,30.032,155.303
C08441=1076.765,365.599,400.199,175.768,30.026,155.302
C08442=1076.760,365.352,400.236,175.765,30.020,155.301
C08443=1076.753,365.104,400.272,175.761,30.014,155.299
C08444=1076.747,364.858,400.310,175.757,30.007,155.298
C08445=1076.741,364.611,400.347,175.754,30.001,155.297
C08446=1076.734,364.363,400.383,175.750,29.995,155.296
C08447=1076.728,364.116,400.420,175.747,29.989,155.295
C08448=1076.722,363.869,400.456,175.743,29.983,155.294
C08449=1076.716,363.621,400.493,175.739,29.977,155.292
C08450=1076.709,363.374,400.531,175.736,29.971,155.291
C08451=1076.702,363.127,400.567,175.732,29.965,155.290
C08452=1076.696,362.880,400.604,175.729,29.959,155.289
C08453=1076.690,362.633,400.640,175.725,29.953,155.288
C08454=1076.683,362.386,400.677,175.721,29.947,155.287
C08455=1076.678,362.139,400.714,175.718,29.941,155.286
C08456=1076.671,361.891,400.750,175.715,29.935,155.284
C08457=1076.664,361.644,400.787,175.710,29.930,155.283
C08458=1076.658,361.397,400.823,175.707,29.924,155.282
C08459=1076.652,361.150,400.860,175.704,29.918,155.281
C08460=1076.645,360.903,400.896,175.700,29.912,155.280
C08461=1076.639,360.656,400.933,175.697,29.906,155.279
C08462=1076.633,360.408,400.968,175.693,29.900,155.278
C08463=1076.628,360.161,401.005,175.689,29.894,155.277
C08464=1076.621,359.914,401.042,175.686,29.888,155.276
C08465=1076.614,359.666,401.079,175.682,29.883,155.275
C08466=1076.608,359.419,401.115,175.679,29.877,155.273
C08467=1076.602,359.171,401.151,175.676,29.871,155.272
C08468=1076.596,358.924,401.187,175.671,29.865,155.271
C08469=1076.590,358.710,401.219,175.669,29.860,155.270
C08470=1076.585,358.497,401.250,175.665,29.855,155.269
C08471=1076.579,358.283,401.281,175.663,29.850,155.268
C08472=1076.574,358.070,401.312,175.659,29.845,155.268
C08473=1076.568,357.856,401.344,175.657,29.840,155.267
C08474=1076.563,357.643,401.375,175.654,29.835,155.266
C08475=1076.558,357.429,401.406,175.650,29.830,155.265
C08476=1076.552,357.215,401.437,175.648,29.825,155.264
C08477=1076.546,356.968,401.474,175.644,29.820,155.263
C08478=1076.540,356.721,401.509,175.641,29.814,155.262
C08479=1076.533,356.474,401.545,175.636,29.808,155.261
C08480=1076.526,356.226,401.581,175.633,29.802,155.260
C08481=1076.520,355.979,401.617,175.630,29.797,155.258
C08482=1076.514,355.731,401.653,175.626,29.791,155.257
C08483=1076.508,355.484,401.690,175.623,29.786,155.256
C08484=1076.502,355.237,401.725,175.620,29.780,155.255
C08485=1076.495,354.990,401.762,175.616,29.774,155.254
C08486=1076.489,354.742,401.798,175.613,29.768,155.253
C08487=1076.483,354.495,401.834,175.609,29.763,155.252
C08488=1076.477,354.248,401.869,175.605,29.757,155.251
C08489=1076.471,354.001,401.905,175.602,29.752,155.250
C08490=1076.465,353.754,401.941,175.598,29.746,155.249
C08491=1076.458,353.506,401.977,175.595,29.741,155.248
C08492=1076.452,353.258,402.012,175.592,29.735,155.247
C08493=1076.445,353.011,402.048,175.588,29.729,155.246
C08494=1076.439,352.764,402.084,175.585,29.724,155.245
C08495=1076.433,352.516,402.120,175.582,29.718,155.244
C08496=1076.427,352.268,402.155,175.578,29.713,155.243
C08497=1076.421,352.022,402.190,175.575,29.707,155.242
C08498=1076.415,351.775,402.227,175.572,29.702,155.241
C08499=1076.409,351.527,402.262,175.567,29.696,155.240
C08500=1076.402,351.280,402.298,175.564,29.690,155.239
C08501=1076.396,351.032,402.333,175.560,29.685,155.238
C08502=1076.390,350.784,402.369,175.557,29.680,155.237
C08503=1076.383,350.537,402.404,175.554,29.674,155.236
C08504=1076.378,350.290,402.439,175.550,29.669,155.235
C08505=1076.371,350.043,402.475,175.547,29.663,155.234
C08506=1076.365,349.795,402.510,175.544,29.658,155.233
C08507=1076.359,349.547,402.546,175.540,29.652,155.232
C08508=1076.352,349.300,402.581,175.537,29.647,155.231
C08509=1076.346,349.046,402.618,175.534,29.641,155.230
C08510=1076.340,348.792,402.653,175.530,29.636,155.229
C08511=1076.334,348.538,402.691,175.527,29.631,155.228
C08512=1076.328,348.284,402.726,175.523,29.625,155.227
C08513=1076.321,348.037,402.762,175.519,29.619,155.226
C08514=1076.315,347.789,402.797,175.516,29.614,155.225
C08515=1076.308,347.542,402.832,175.512,29.609,155.224
C08516=1076.303,347.295,402.868,175.509,29.603,155.223
C08517=1076.296,347.047,402.902,175.506,29.598,155.222
C08518=1076.290,346.799,402.938,175.502,29.593,155.221
C08519=1076.284,346.552,402.973,175.499,29.587,155.220
C08520=1076.278,346.305,403.008,175.496,29.582,155.219
C08521=1076.271,346.057,403.044,175.492,29.577,155.218
C08522=1076.265,345.809,403.079,175.489,29.571,155.217
C08523=1076.259,345.562,403.113,175.486,29.566,155.216
C08524=1076.253,345.315,403.149,175.482,29.561,155.215
C08525=1076.243,344.897,403.208,175.477,29.552,155.214
C08526=1076.233,344.481,403.267,175.471,29.543,155.212
C08527=1076.222,344.063,403.325,175.465,29.534,155.210
C08528=1076.212,343.646,403.384,175.460,29.526,155.209
C08529=1076.205,343.398,403.419,175.457,29.521,155.208
C08530=1076.200,343.151,403.454,175.454,29.515,155.207
C08531=1076.193,342.903,403.489,175.450,29.510,155.206
C08532=1076.186,342.656,403.524,175.447,29.505,155.205
C08533=1076.181,342.408,403.558,175.444,29.500,155.204
C08534=1076.174,342.161,403.593,175.440,29.495,155.203
C08535=1076.169,341.913,403.628,175.437,29.490,155.202
C08536=1076.162,341.666,403.663,175.433,29.485,155.201
C08537=1076.155,341.418,403.697,175.430,29.479,155.200
C08538=1076.150,341.170,403.732,175.427,29.474,155.200
C08539=1076.144,340.923,403.767,175.423,29.469,155.199
C08540=1076.138,340.676,403.801,175.420,29.464,155.198
C08541=1076.131,340.428,403.835,175.417,29.459,155.197
C08542=1076.125,340.181,403.870,175.414,29.454,155.196
C08543=1076.119,339.933,403.905,175.411,29.449,155.195
C08544=1076.113,339.685,403.939,175.407,29.444,155.194
C08545=1076.107,339.437,403.974,175.404,29.439,155.193
C08546=1076.101,339.191,404.008,175.401,29.433,155.192
C08547=1076.094,338.943,404.043,175.397,29.428,155.191
C08548=1076.089,338.695,404.077,175.394,29.423,155.190
C08549=1076.083,338.447,404.112,175.391,29.418,155.190
C08550=1076.077,338.200,404.146,175.387,29.413,155.189
C08551=1076.070,337.952,404.180,175.384,29.408,155.188
C08552=1076.065,337.705,404.214,175.382,29.403,155.187
C08553=1076.058,337.457,404.249,175.378,29.398,155.186
C08554=1076.052,337.210,404.284,175.375,29.393,155.185
C08555=1076.045,336.962,404.318,175.371,29.388,155.184
C08556=1076.040,336.715,404.352,175.368,29.383,155.183
C08557=1076.033,336.467,404.386,175.365,29.378,155.183
C08558=1076.027,336.220,404.420,175.361,29.373,155.182
C08559=1076.021,335.972,404.455,175.358,29.368,155.181
C08560=1076.015,335.724,404.489,175.356,29.363,155.180
C08561=1076.009,335.477,404.523,175.352,29.358,155.179
C08562=1076.003,335.229,404.557,175.349,29.353,155.178
C08563=1075.997,334.981,404.591,175.345,29.348,155.177
C08564=1075.991,334.733,404.625,175.342,29.343,155.176
C08565=1075.985,334.486,404.659,175.339,29.338,155.175
C08566=1075.979,334.239,404.693,175.335,29.334,155.175
C08567=1075.972,333.991,404.728,175.333,29.329,155.174
C08568=1075.967,333.743,404.762,175.330,29.324,155.173
C08569=1075.961,333.496,404.796,175.326,29.319,155.172
C08570=1075.954,333.248,404.829,175.323,29.314,155.171
C08571=1075.948,333.000,404.863,175.320,29.309,155.170
C08572=1075.942,332.753,404.897,175.316,29.304,155.169
C08573=1075.936,332.505,404.931,175.314,29.299,155.169
C08574=1075.930,332.257,404.965,175.310,29.294,155.168
C08575=1075.924,332.010,404.999,175.307,29.290,155.167
C08576=1075.918,331.762,405.033,175.304,29.285,155.166
C08577=1075.913,331.548,405.062,175.301,29.280,155.165
C08578=1075.907,331.333,405.092,175.299,29.276,155.165
C08579=1075.903,331.119,405.121,175.295,29.272,155.164
C08580=1075.897,330.904,405.150,175.293,29.268,155.163
C08581=1075.891,330.689,405.179,175.290,29.264,155.162
C08582=1075.886,330.475,405.208,175.287,29.259,155.162
C08583=1075.881,330.260,405.237,175.284,29.256,155.161
C08584=1075.875,330.045,405.267,175.282,29.252,155.160
C08585=1075.869,329.798,405.300,175.279,29.247,155.159
C08586=1075.863,329.551,405.333,175.275,29.242,155.159
C08587=1075.857,329.302,405.367,175.272,29.237,155.158
C08588=1075.850,329.055,405.401,175.269,29.233,155.157
C08589=1075.844,328.807,405.434,175.266,29.228,155.156
C08590=1075.837,328.559,405.468,175.263,29.223,155.155
C08591=1075.832,328.311,405.501,175.259,29.218,155.155
C08592=1075.826,328.064,405.535,175.256,29.214,155.154
C08593=1075.819,327.817,405.568,175.253,29.209,155.153
C08594=1075.813,327.568,405.602,175.250,29.204,155.152
C08595=1075.807,327.321,405.635,175.247,29.200,155.151
C08596=1075.801,327.073,405.668,175.243,29.195,155.151
C08597=1075.795,326.826,405.701,175.241,29.191,155.150
C08598=1075.788,326.578,405.735,175.238,29.185,155.149
C08599=1075.782,326.330,405.768,175.234,29.181,155.148
C08600=1075.777,326.082,405.802,175.231,29.176,155.147
C08601=1075.770,325.835,405.835,175.228,29.172,155.146
C08602=1075.764,325.587,405.868,175.225,29.167,155.146
C08603=1075.758,325.340,405.901,175.222,29.162,155.145
C08604=1075.752,325.091,405.935,175.218,29.158,155.144
C08605=1075.745,324.844,405.968,175.216,29.153,155.143
C08606=1075.740,324.596,406.002,175.213,29.149,155.143
C08607=1075.734,324.349,406.034,175.209,29.143,155.142
C08608=1075.728,324.101,406.068,175.206,29.139,155.141
C08609=1075.722,323.853,406.100,175.203,29.134,155.140
C08610=1075.716,323.605,406.134,175.200,29.130,155.139
C08611=1075.710,323.358,406.166,175.197,29.125,155.139
C08612=1075.703,323.109,406.200,175.194,29.121,155.138
C08613=1075.697,322.862,406.234,175.191,29.116,155.137
C08614=1075.691,322.614,406.266,175.188,29.111,155.136
C08615=1075.685,322.366,406.300,175.184,29.106,155.135
C08616=1075.679,322.119,406.332,175.182,29.102,155.134
C08617=1075.673,321.871,406.366,175.178,29.097,155.134
C08618=1075.667,321.623,406.399,175.175,29.093,155.133
C08619=1075.661,321.376,406.431,175.173,29.088,155.132
C08620=1075.655,321.128,406.465,175.169,29.084,155.131
C08621=1075.649,320.880,406.497,175.166,29.079,155.131
C08622=1075.644,320.632,406.530,175.164,29.075,155.130
C08623=1075.637,320.384,406.563,175.160,29.070,155.129
C08624=1075.631,320.137,406.595,175.157,29.065,155.128
C08625=1075.626,319.889,406.629,175.154,29.061,155.127
C08626=1075.619,319.641,406.662,175.151,29.056,155.127
C08627=1075.614,319.393,406.695,175.148,29.051,155.126
C08628=1075.607,319.146,406.728,175.145,29.047,155.125
C08629=1075.601,318.898,406.760,175.142,29.042,155.124
C08630=1075.596,318.650,406.793,175.139,29.038,155.124
C08631=1075.590,318.403,406.825,175.136,29.033,155.123
C08632=1075.584,318.155,406.858,175.133,29.029,155.122
C08633=1075.579,317.937,406.887,175.130,29.025,155.121
C08634=1075.573,317.719,406.916,175.127,29.021,155.121
C08635=1075.568,317.501,406.944,175.124,29.017,155.120
C08636=1075.563,317.284,406.973,175.122,29.012,155.119
C08637=1075.558,317.065,407.002,175.120,29.009,155.119
C08638=1075.553,316.848,407.031,175.117,29.005,155.118
C08639=1075.548,316.630,407.060,175.114,29.001,155.117
C08640=1075.543,316.413,407.088,175.111,28.997,155.117
C08641=1075.537,316.164,407.120,175.109,28.992,155.116
C08642=1075.531,315.917,407.153,175.105,28.988,155.115
C08643=1075.525,315.669,407.186,175.102,28.983,155.114
C08644=1075.519,315.421,407.219,175.100,28.979,155.113
C08645=1075.514,315.174,407.251,175.096,28.974,155.113
C08646=1075.508,314.926,407.283,175.094,28.970,155.112
C08647=1075.502,314.678,407.316,175.091,28.965,155.111
C08648=1075.496,314.429,407.348,175.087,28.960,155.110
C08649=1075.490,314.182,407.381,175.085,28.956,155.110
C08650=1075.483,313.934,407.413,175.082,28.952,155.109
C08651=1075.477,313.686,407.445,175.078,28.947,155.108
C08652=1075.471,313.439,407.477,175.076,28.943,155.108
C08653=1075.465,313.191,407.510,175.072,28.939,155.107
C08654=1075.459,312.943,407.542,175.070,28.935,155.106
C08655=1075.453,312.695,407.574,175.067,28.930,155.105
C08656=1075.447,312.447,407.606,175.063,28.925,155.105
C08657=1075.440,312.199,407.638,175.061,28.921,155.104
C08658=1075.434,311.952,407.671,175.057,28.917,155.103
C08659=1075.428,311.704,407.702,175.054,28.913,155.102
C08660=1075.422,311.456,407.734,175.052,28.908,155.102
C08661=1075.416,311.208,407.767,175.048,28.904,155.101
C08662=1075.410,310.960,407.799,175.046,28.900,155.100
C08663=1075.403,310.712,407.831,175.042,28.895,155.100
C08664=1075.398,310.465,407.862,175.039,28.891,155.099
C08665=1075.392,310.217,407.895,175.037,28.887,155.098
C08666=1075.386,309.969,407.927,175.033,28.882,155.097
C08667=1075.380,309.721,407.959,175.031,28.878,155.097
C08668=1075.374,309.474,407.990,175.028,28.873,155.096
C08669=1075.368,309.225,408.022,175.024,28.869,155.095
C08670=1075.361,308.978,408.055,175.022,28.865,155.094
C08671=1075.355,308.730,408.087,175.018,28.861,155.094
C08672=1075.349,308.482,408.118,175.016,28.856,155.093
C08673=1075.343,308.234,408.150,175.013,28.852,155.092
C08674=1075.337,307.986,408.182,175.010,28.848,155.092
C08675=1075.332,307.738,408.214,175.007,28.844,155.091
C08676=1075.325,307.491,408.245,175.004,28.839,155.090
C08677=1075.319,307.242,408.277,175.001,28.835,155.090
C08678=1075.314,306.995,408.309,174.998,28.830,155.089
C08679=1075.308,306.747,408.341,174.995,28.826,155.088
C08680=1075.301,306.499,408.373,174.992,28.822,155.087
C08681=1075.295,306.252,408.405,174.990,28.818,155.087
C08682=1075.289,306.004,408.437,174.986,28.813,155.086
C08683=1075.284,305.755,408.468,174.983,28.809,155.085
C08684=1075.278,305.508,408.499,174.980,28.805,155.085
C08685=1075.272,305.259,408.531,174.977,28.800,155.084
C08686=1075.266,305.012,408.563,174.975,28.796,155.083
C08687=1075.260,304.764,408.594,174.971,28.792,155.082
C08688=1075.254,304.516,408.626,174.969,28.787,155.082
C08689=1075.249,304.300,408.654,174.966,28.784,155.081
C08690=1075.244,304.084,408.681,174.964,28.780,155.080
C08691=1075.239,303.867,408.709,174.961,28.776,155.080
C08692=1075.233,303.651,408.736,174.958,28.773,155.079
C08693=1075.228,303.435,408.764,174.956,28.769,155.079
C08694=1075.223,303.219,408.791,174.953,28.765,155.078
C08695=1075.218,303.003,408.819,174.951,28.761,155.077
C08696=1075.213,302.787,408.846,174.948,28.758,155.077
C08697=1075.207,302.539,408.878,174.946,28.754,155.076
C08698=1075.201,302.291,408.910,174.943,28.749,155.075
C08699=1075.196,302.043,408.940,174.940,28.745,155.075
C08700=1075.190,301.796,408.972,174.937,28.740,155.074
C08701=1075.184,301.547,409.004,174.933,28.736,155.073
C08702=1075.177,301.300,409.035,174.931,28.732,155.073
C08703=1075.172,301.051,409.066,174.928,28.728,155.072
C08704=1075.166,300.804,409.098,174.925,28.723,155.071
C08705=1075.160,300.556,409.129,174.922,28.719,155.070
C08706=1075.155,300.308,409.160,174.920,28.715,155.070
C08707=1075.149,300.060,409.192,174.916,28.710,155.069
C08708=1075.143,299.812,409.222,174.914,28.706,155.068
C08709=1075.137,299.564,409.254,174.911,28.702,155.068
C08710=1075.131,299.316,409.285,174.908,28.698,155.067
C08711=1075.126,299.068,409.316,174.906,28.693,155.066
C08712=1075.119,298.820,409.348,174.902,28.689,155.066
C08713=1075.114,298.572,409.379,174.900,28.685,155.065
C08714=1075.108,298.325,409.410,174.897,28.681,155.064
C08715=1075.102,298.076,409.441,174.894,28.677,155.063
C08716=1075.097,297.829,409.473,174.891,28.672,155.063
C08717=1075.091,297.581,409.503,174.889,28.668,155.062
C08718=1075.085,297.333,409.535,174.885,28.664,155.061
C08719=1075.079,297.085,409.566,174.883,28.659,155.061
C08720=1075.073,296.836,409.596,174.879,28.655,155.060
C08721=1075.067,296.589,409.628,174.877,28.651,155.059
C08722=1075.061,296.340,409.659,174.874,28.647,155.059
C08723=1075.055,296.093,409.690,174.871,28.643,155.058
C08724=1075.050,295.845,409.721,174.868,28.639,155.057
C08725=1075.043,295.596,409.751,174.866,28.635,155.057
C08726=1075.037,295.349,409.782,174.863,28.631,155.056
C08727=1075.031,295.101,409.813,174.860,28.627,155.055
C08728=1075.025,294.853,409.844,174.857,28.623,155.055
C08729=1075.020,294.605,409.874,174.854,28.618,155.054
C08730=1075.013,294.357,409.906,174.852,28.614,155.053
C08731=1075.007,294.109,409.936,174.848,28.610,155.053
C08732=1075.002,293.861,409.967,174.846,28.606,155.052
C08733=1074.996,293.612,409.998,174.842,28.602,155.051
C08734=1074.990,293.365,410.028,174.840,28.598,155.051
C08735=1074.984,293.117,410.059,174.838,28.593,155.050
C08736=1074.977,292.869,410.090,174.834,28.589,155.049
C08737=1074.972,292.621,410.121,174.832,28.585,155.049
C08738=1074.966,292.373,410.151,174.829,28.581,155.048
C08739=1074.961,292.125,410.182,174.826,28.577,155.047
C08740=1074.954,291.876,410.212,174.823,28.573,155.047
C08741=1074.948,291.629,410.243,174.820,28.569,155.046
C08742=1074.942,291.381,410.273,174.818,28.565,155.045
C08743=1074.937,291.132,410.304,174.815,28.560,155.045
C08744=1074.931,290.884,410.335,174.812,28.556,155.044
C08745=1074.921,290.467,410.386,174.807,28.550,155.043
C08746=1074.911,290.049,410.438,174.802,28.543,155.042
C08747=1074.901,289.631,410.489,174.798,28.536,155.041
C08748=1074.891,289.214,410.540,174.794,28.529,155.040
C08749=1074.885,288.966,410.570,174.790,28.525,155.039
C08750=1074.879,288.718,410.601,174.788,28.521,155.038
C08751=1074.873,288.470,410.631,174.785,28.517,155.038
C08752=1074.867,288.222,410.662,174.782,28.513,155.037
C08753=1074.861,287.973,410.692,174.780,28.509,155.036
C08754=1074.855,287.725,410.722,174.776,28.505,155.036
C08755=1074.849,287.477,410.752,174.774,28.501,155.035
C08756=1074.844,287.229,410.783,174.772,28.497,155.034
C08757=1074.838,286.981,410.813,174.768,28.492,155.034
C08758=1074.831,286.733,410.843,174.766,28.488,155.033
C08759=1074.825,286.485,410.873,174.763,28.485,155.032
C08760=1074.819,286.237,410.903,174.760,28.480,155.032
C08761=1074.814,285.989,410.934,174.758,28.476,155.031
C08762=1074.808,285.741,410.963,174.754,28.472,155.030
C08763=1074.802,285.492,410.994,174.752,28.468,155.030
C08764=1074.796,285.244,411.024,174.750,28.464,155.029
C08765=1074.790,284.997,411.055,174.746,28.460,155.029
C08766=1074.784,284.748,411.084,174.744,28.456,155.028
C08767=1074.778,284.501,411.114,174.741,28.452,155.027
C08768=1074.772,284.253,411.144,174.738,28.448,155.027
C08769=1074.767,284.004,411.174,174.736,28.444,155.026
C08770=1074.761,283.757,411.204,174.733,28.440,155.025
C08771=1074.755,283.507,411.234,174.730,28.436,155.025
C08772=1074.749,283.260,411.265,174.728,28.432,155.024
C08773=1074.743,283.011,411.294,174.725,28.428,155.023
C08774=1074.737,282.764,411.324,174.722,28.424,155.023
C08775=1074.731,282.516,411.355,174.719,28.420,155.022
C08776=1074.725,282.267,411.384,174.717,28.416,155.021
C08777=1074.720,282.020,411.414,174.714,28.412,155.021
C08778=1074.714,281.771,411.444,174.711,28.408,155.020
C08779=1074.708,281.523,411.474,174.709,28.404,155.019
C08780=1074.702,281.275,411.504,174.706,28.400,155.019
C08781=1074.697,281.027,411.533,174.703,28.396,155.018
C08782=1074.691,280.779,411.564,174.701,28.392,155.018
C08783=1074.685,280.530,411.593,174.697,28.388,155.017
C08784=1074.679,280.283,411.623,174.695,28.384,155.016
C08785=1074.673,280.034,411.653,174.693,28.380,155.016
C08786=1074.668,279.786,411.682,174.689,28.376,155.015
C08787=1074.660,279.538,411.712,174.687,28.372,155.014
C08788=1074.655,279.289,411.742,174.685,28.368,155.014
C08789=1074.649,279.041,411.771,174.681,28.364,155.013
C08790=1074.643,278.793,411.801,174.679,28.360,155.013
C08791=1074.637,278.545,411.831,174.676,28.356,155.012
C08792=1074.631,278.297,411.860,174.673,28.352,155.011
C08793=1074.625,278.049,411.890,174.671,28.348,155.011
C08794=1074.620,277.801,411.920,174.668,28.344,155.010
C08795=1074.614,277.552,411.949,174.665,28.340,155.009
C08796=1074.608,277.304,411.979,174.663,28.336,155.009
C08797=1074.598,276.897,412.027,174.659,28.330,155.008
C08798=1074.589,276.489,412.076,174.654,28.323,155.007
C08799=1074.579,276.081,412.124,174.650,28.316,155.006
C08800=1074.570,275.674,412.172,174.646,28.310,155.005
C08801=1074.564,275.425,412.201,174.642,28.306,155.004
C08802=1074.558,275.178,412.231,174.640,28.302,155.003
C08803=1074.552,274.930,412.261,174.638,28.298,155.003
C08804=1074.546,274.681,412.290,174.634,28.294,155.002
C08805=1074.540,274.433,412.319,174.632,28.290,155.001
C08806=1074.534,274.185,412.348,174.630,28.287,155.001
C08807=1074.528,273.936,412.378,174.627,28.283,155.000
C08808=1074.522,273.688,412.407,174.624,28.278,155.000
C08809=1074.517,273.440,412.437,174.621,28.274,154.999
C08810=1074.510,273.192,412.466,174.619,28.270,154.998
C08811=1074.505,272.943,412.495,174.617,28.266,154.998
C08812=1074.499,272.696,412.524,174.613,28.263,154.997
C08813=1074.493,272.448,412.553,174.611,28.259,154.997
C08814=1074.488,272.199,412.582,174.609,28.255,154.996
C08815=1074.482,271.950,412.611,174.606,28.251,154.995
C08816=1074.475,271.702,412.640,174.603,28.247,154.995
C08817=1074.470,271.454,412.670,174.601,28.243,154.994
C08818=1074.464,271.206,412.699,174.598,28.239,154.993
C08819=1074.457,270.958,412.728,174.596,28.235,154.993
C08820=1074.452,270.710,412.757,174.593,28.231,154.992
C08821=1074.446,270.462,412.786,174.590,28.227,154.992
C08822=1074.440,270.213,412.814,174.588,28.223,154.991
C08823=1074.435,269.965,412.844,174.585,28.220,154.990
C08824=1074.428,269.716,412.873,174.582,28.215,154.990
C08825=1074.422,269.468,412.902,174.580,28.212,154.989
C08826=1074.418,269.220,412.931,174.577,28.208,154.989
C08827=1074.411,268.972,412.960,174.575,28.204,154.988
C08828=1074.405,268.724,412.989,174.572,28.200,154.987
C08829=1074.399,268.476,413.018,174.569,28.196,154.987
C08830=1074.393,268.227,413.046,174.567,28.192,154.986
C08831=1074.387,267.978,413.076,174.564,28.188,154.985
C08832=1074.382,267.731,413.104,174.561,28.184,154.985
C08833=1074.376,267.482,413.133,174.559,28.181,154.984
C08834=1074.370,267.234,413.162,174.556,28.177,154.984
C08835=1074.364,266.985,413.190,174.554,28.173,154.983
C08836=1074.359,266.738,413.219,174.552,28.169,154.982
C08837=1074.352,266.489,413.248,174.548,28.165,154.982
C08838=1074.347,266.241,413.277,174.546,28.161,154.981
C08839=1074.340,265.993,413.306,174.544,28.157,154.981
C08840=1074.335,265.744,413.334,174.541,28.153,154.980
C08841=1074.329,265.496,413.363,174.539,28.149,154.979
C08842=1074.324,265.247,413.392,174.536,28.145,154.979
C08843=1074.317,264.999,413.421,174.533,28.141,154.978
C08844=1074.312,264.751,413.449,174.531,28.137,154.977
C08845=1074.306,264.503,413.478,174.528,28.134,154.977
C08846=1074.300,264.254,413.506,174.526,28.130,154.976
C08847=1074.294,264.007,413.535,174.523,28.125,154.976
C08848=1074.288,263.758,413.563,174.520,28.121,154.975
C08849=1074.278,263.354,413.610,174.516,28.115,154.974
C08850=1074.268,262.949,413.656,174.512,28.109,154.973
C08851=1074.259,262.545,413.702,174.508,28.103,154.972
C08852=1074.249,262.140,413.748,174.504,28.097,154.971
C08853=1074.243,261.892,413.777,174.501,28.093,154.971
C08854=1074.237,261.643,413.805,174.499,28.089,154.970
C08855=1074.231,261.395,413.833,174.496,28.085,154.969
C08856=1074.225,261.147,413.862,174.494,28.082,154.969
C08857=1074.219,260.898,413.891,174.491,28.078,154.968
C08858=1074.213,260.650,413.918,174.488,28.074,154.968
C08859=1074.207,260.402,413.946,174.486,28.070,154.967
C08860=1074.201,260.153,413.975,174.484,28.066,154.966
C08861=1074.196,259.905,414.003,174.481,28.063,154.966
C08862=1074.190,259.657,414.032,174.479,28.059,154.965
C08863=1074.183,259.408,414.059,174.475,28.055,154.965
C08864=1074.178,259.160,414.087,174.473,28.051,154.964
C08865=1074.171,258.912,414.116,174.471,28.047,154.963
C08866=1074.165,258.663,414.145,174.468,28.043,154.963
C08867=1074.160,258.415,414.173,174.466,28.039,154.962
C08868=1074.153,258.167,414.200,174.464,28.035,154.962
C08869=1074.148,257.918,414.229,174.460,28.032,154.961
C08870=1074.142,257.670,414.257,174.458,28.028,154.960
C08871=1074.136,257.421,414.285,174.456,28.024,154.960
C08872=1074.131,257.173,414.313,174.453,28.020,154.959
C08873=1074.124,256.925,414.341,174.451,28.016,154.959
C08874=1074.118,256.676,414.369,174.449,28.013,154.958
C08875=1074.113,256.428,414.397,174.446,28.009,154.957
C08876=1074.107,256.179,414.425,174.443,28.004,154.957
C08877=1074.101,255.931,414.453,174.441,28.001,154.956
C08878=1074.095,255.683,414.481,174.438,27.997,154.956
C08879=1074.090,255.435,414.509,174.436,27.993,154.955
C08880=1074.084,255.186,414.537,174.433,27.989,154.954
C08881=1074.078,254.938,414.565,174.431,27.985,154.954
C08882=1074.072,254.689,414.593,174.429,27.981,154.953
C08883=1074.066,254.441,414.621,174.426,27.978,154.953
C08884=1074.060,254.193,414.649,174.423,27.974,154.952
C08885=1074.054,253.944,414.677,174.421,27.970,154.951
C08886=1074.048,253.696,414.705,174.418,27.966,154.951
C08887=1074.042,253.447,414.733,174.416,27.962,154.950
C08888=1074.037,253.199,414.760,174.414,27.958,154.950
C08889=1074.031,252.951,414.788,174.411,27.955,154.949
C08890=1074.025,252.702,414.816,174.409,27.951,154.948
C08891=1074.019,252.454,414.844,174.407,27.947,154.948
C08892=1074.013,252.206,414.872,174.404,27.943,154.947
C08893=1074.008,251.957,414.899,174.401,27.939,154.947
C08894=1074.002,251.709,414.927,174.399,27.935,154.946
C08895=1073.996,251.461,414.955,174.396,27.931,154.945
C08896=1073.990,251.212,414.983,174.394,27.927,154.945
C08897=1073.985,250.963,415.010,174.392,27.923,154.944
C08898=1073.979,250.715,415.038,174.389,27.920,154.944
C08899=1073.973,250.467,415.066,174.387,27.916,154.943
C08900=1073.967,250.219,415.093,174.385,27.912,154.942
C08901=1073.958,249.811,415.138,174.381,27.906,154.941
C08902=1073.949,249.404,415.184,174.377,27.899,154.940
C08903=1073.939,248.997,415.229,174.373,27.893,154.939
C08904=1073.930,248.590,415.274,174.369,27.887,154.938
C08905=1073.924,248.342,415.302,174.367,27.883,154.938
C08906=1073.919,248.093,415.330,174.363,27.878,154.937
C08907=1073.913,247.845,415.357,174.361,27.874,154.937
C08908=1073.907,247.596,415.384,174.359,27.871,154.936
C08909=1073.902,247.348,415.413,174.356,27.867,154.935
C08910=1073.896,247.099,415.439,174.354,27.863,154.935
C08911=1073.890,246.851,415.467,174.352,27.859,154.934
C08912=1073.884,246.602,415.494,174.349,27.855,154.934
C08913=1073.879,246.354,415.522,174.347,27.851,154.933
C08914=1073.873,246.106,415.549,174.345,27.847,154.932
C08915=1073.866,245.857,415.577,174.342,27.844,154.932
C08916=1073.861,245.609,415.604,174.340,27.840,154.931
C08917=1073.855,245.361,415.631,174.338,27.836,154.931
C08918=1073.849,245.112,415.659,174.335,27.832,154.930
C08919=1073.844,244.863,415.686,174.333,27.828,154.929
C08920=1073.838,244.615,415.713,174.331,27.825,154.929
C08921=1073.833,244.367,415.740,174.328,27.821,154.928
C08922=1073.826,244.118,415.768,174.326,27.817,154.927
C08923=1073.821,243.870,415.795,174.323,27.813,154.927
C08924=1073.815,243.621,415.822,174.320,27.809,154.926
C08925=1073.808,243.373,415.850,174.318,27.805,154.926
C08926=1073.803,243.124,415.877,174.316,27.801,154.925
C08927=1073.798,242.876,415.903,174.313,27.797,154.925
C08928=1073.792,242.627,415.930,174.311,27.793,154.924
C08929=1073.786,242.379,415.958,174.309,27.790,154.923
C08930=1073.780,242.130,415.985,174.306,27.786,154.923
C08931=1073.774,241.882,416.012,174.304,27.782,154.922
C08932=1073.768,241.633,416.039,174.302,27.778,154.922
C08933=1073.762,241.385,416.066,174.299,27.774,154.921
C08934=1073.757,241.137,416.093,174.297,27.771,154.920
C08935=1073.751,240.888,416.120,174.295,27.767,154.920
C08936=1073.745,240.639,416.147,174.292,27.763,154.919
C08937=1073.739,240.391,416.174,174.290,27.759,154.919
C08938=1073.733,240.142,416.200,174.288,27.755,154.918
C08939=1073.727,239.895,416.228,174.285,27.751,154.917
C08940=1073.721,239.645,416.255,174.283,27.747,154.917
C08941=1073.716,239.397,416.282,174.281,27.743,154.916
C08942=1073.710,239.149,416.309,174.278,27.740,154.916
C08943=1073.704,238.900,416.335,174.276,27.736,154.915
C08944=1073.698,238.651,416.362,174.274,27.732,154.914
C08945=1073.692,238.403,416.389,174.272,27.728,154.914
C08946=1073.686,238.154,416.416,174.269,27.724,154.913
C08947=1073.680,237.906,416.442,174.267,27.721,154.913
C08948=1073.675,237.658,416.469,174.265,27.717,154.912
C08949=1073.669,237.408,416.496,174.262,27.713,154.911
C08950=1073.663,237.160,416.523,174.260,27.709,154.911
C08951=1073.657,236.912,416.550,174.258,27.705,154.910
C08952=1073.652,236.663,416.576,174.255,27.702,154.910
C08953=1073.642,236.249,416.621,174.251,27.695,154.909
C08954=1073.633,235.836,416.665,174.248,27.689,154.908
C08955=1073.622,235.423,416.709,174.244,27.682,154.907
C08956=1073.613,235.009,416.754,174.240,27.676,154.906
C08957=1073.607,234.761,416.781,174.237,27.672,154.905
C08958=1073.601,234.512,416.807,174.235,27.668,154.904
C08959=1073.596,234.263,416.833,174.233,27.664,154.904
C08960=1073.590,234.015,416.860,174.231,27.660,154.903
C08961=1073.585,233.766,416.887,174.228,27.656,154.903
C08962=1073.578,233.518,416.913,174.226,27.652,154.902
C08963=1073.572,233.268,416.939,174.224,27.649,154.902
C08964=1073.566,233.020,416.966,174.221,27.645,154.901
C08965=1073.561,232.772,416.993,174.219,27.641,154.900
C08966=1073.555,232.523,417.019,174.217,27.637,154.900
C08967=1073.549,232.274,417.045,174.214,27.633,154.899
C08968=1073.544,232.026,417.072,174.212,27.629,154.898
C08969=1073.538,231.778,417.099,174.210,27.626,154.898
C08970=1073.532,231.529,417.125,174.207,27.622,154.897
C08971=1073.527,231.280,417.151,174.206,27.618,154.897
C08972=1073.521,231.032,417.178,174.204,27.614,154.896
C08973=1073.515,230.784,417.204,174.202,27.610,154.895
C08974=1073.509,230.535,417.230,174.199,27.607,154.895
C08975=1073.503,230.287,417.256,174.197,27.603,154.894
C08976=1073.497,230.038,417.283,174.195,27.599,154.894
C08977=1073.492,229.789,417.309,174.192,27.595,154.893
C08978=1073.486,229.541,417.336,174.190,27.591,154.893
C08979=1073.479,229.292,417.361,174.188,27.587,154.892
C08980=1073.473,229.043,417.388,174.185,27.583,154.891
C08981=1073.468,228.794,417.414,174.183,27.579,154.891
C08982=1073.462,228.546,417.441,174.181,27.576,154.890
C08983=1073.456,228.297,417.466,174.178,27.572,154.890
C08984=1073.450,228.049,417.493,174.176,27.568,154.889
C08985=1073.445,227.800,417.519,174.174,27.564,154.888
C08986=1073.438,227.552,417.545,174.172,27.560,154.888
C08987=1073.433,227.303,417.571,174.169,27.557,154.887
C08988=1073.427,227.054,417.597,174.167,27.553,154.887
C08989=1073.421,226.806,417.623,174.166,27.549,154.886
C08990=1073.415,226.557,417.649,174.163,27.545,154.885
C08991=1073.410,226.308,417.675,174.161,27.541,154.885
C08992=1073.403,226.060,417.701,174.159,27.538,154.884
C08993=1073.398,225.811,417.727,174.156,27.534,154.884
C08994=1073.392,225.562,417.753,174.154,27.529,154.883
C08995=1073.386,225.315,417.779,174.152,27.526,154.882
C08996=1073.381,225.066,417.805,174.149,27.522,154.882
C08997=1073.375,224.818,417.831,174.147,27.518,154.881
C08998=1073.369,224.569,417.857,174.145,27.514,154.881
C08999=1073.363,224.320,417.883,174.143,27.510,154.880
C09000=1073.358,224.072,417.909,174.141,27.506,154.879
C09001=1073.351,223.823,417.935,174.139,27.503,154.879
C09002=1073.346,223.574,417.960,174.137,27.499,154.878
C09003=1073.340,223.325,417.986,174.134,27.495,154.878
C09004=1073.334,223.077,418.012,174.132,27.491,154.877
C09005=1073.329,222.866,418.034,174.130,27.488,154.877
C09006=1073.324,222.655,418.056,174.128,27.484,154.876
C09007=1073.319,222.444,418.078,174.127,27.481,154.875
C09008=1073.315,222.233,418.100,174.125,27.478,154.875
C09009=1073.310,222.023,418.122,174.123,27.475,154.874
C09010=1073.305,221.812,418.144,174.121,27.471,154.874
C09011=1073.300,221.601,418.165,174.119,27.468,154.873
C09012=1073.295,221.390,418.187,174.117,27.465,154.873
C09013=1073.290,221.141,418.213,174.115,27.460,154.872
C09014=1073.284,220.892,418.238,174.113,27.457,154.872
C09015=1073.277,220.643,418.264,174.111,27.453,154.871
C09016=1073.272,220.395,418.290,174.109,27.450,154.871
C09017=1073.265,220.146,418.316,174.106,27.446,154.870
C09018=1073.260,219.897,418.341,174.104,27.441,154.869
C09019=1073.254,219.649,418.367,174.102,27.438,154.869
C09020=1073.248,219.401,418.392,174.100,27.434,154.868
C09021=1073.243,219.152,418.418,174.097,27.430,154.868
C09022=1073.236,218.903,418.443,174.095,27.426,154.867
C09023=1073.231,218.654,418.469,174.094,27.422,154.866
C09024=1073.225,218.406,418.494,174.091,27.419,154.866
C09025=1073.219,218.157,418.520,174.089,27.415,154.865
C09026=1073.214,217.909,418.545,174.087,27.411,154.865
C09027=1073.207,217.660,418.571,174.085,27.407,154.864
C09028=1073.201,217.411,418.596,174.082,27.403,154.863
C09029=1073.196,217.162,418.622,174.080,27.399,154.863
C09030=1073.190,216.914,418.647,174.079,27.396,154.862
C09031=1073.184,216.666,418.672,174.076,27.392,154.862
C09032=1073.179,216.417,418.698,174.074,27.388,154.861
C09033=1073.172,216.168,418.723,174.072,27.384,154.860
C09034=1073.166,215.919,418.749,174.070,27.380,154.860
C09035=1073.161,215.671,418.774,174.067,27.376,154.859
C09036=1073.155,215.422,418.800,174.065,27.372,154.859
C09037=1073.149,215.174,418.825,174.064,27.368,154.858
C09038=1073.144,214.924,418.850,174.061,27.364,154.857
C09039=1073.138,214.676,418.875,174.059,27.360,154.857
C09040=1073.132,214.427,418.901,174.057,27.357,154.856
C09041=1073.126,214.178,418.926,174.055,27.353,154.856
C09042=1073.121,213.931,418.951,174.052,27.349,154.855
C09043=1073.115,213.682,418.977,174.051,27.345,154.854
C09044=1073.109,213.432,419.002,174.049,27.341,154.854
C09045=1073.104,213.184,419.027,174.047,27.337,154.853
C09046=1073.098,212.936,419.052,174.044,27.333,154.852
C09047=1073.091,212.687,419.078,174.042,27.329,154.852
C09048=1073.086,212.437,419.103,174.040,27.325,154.851
C09049=1073.081,212.189,419.128,174.038,27.322,154.851
C09050=1073.074,211.941,419.153,174.036,27.318,154.850
C09051=1073.068,211.692,419.178,174.034,27.314,154.849
C09052=1073.063,211.443,419.203,174.032,27.310,154.849
C09053=1073.057,211.195,419.228,174.029,27.306,154.848
C09054=1073.051,210.946,419.253,174.027,27.302,154.848
C09055=1073.046,210.697,419.278,174.026,27.298,154.847
C09056=1073.040,210.449,419.304,174.024,27.294,154.846
C09057=1073.034,210.200,419.329,174.021,27.291,154.846
C09058=1073.028,209.951,419.353,174.019,27.287,154.845
C09059=1073.022,209.703,419.379,174.017,27.283,154.845
C09060=1073.016,209.453,419.403,174.015,27.279,154.844
C09061=1073.007,209.036,419.445,174.012,27.272,154.843
C09062=1072.997,208.619,419.487,174.008,27.266,154.842
C09063=1072.987,208.201,419.529,174.004,27.259,154.841
C09064=1072.977,207.784,419.571,174.001,27.253,154.840
C09065=1072.953,206.743,419.672,173.874,27.187,154.839
C09066=1072.947,206.494,419.696,173.872,27.184,154.838
C09067=1072.942,206.245,419.721,173.870,27.181,154.838
C09068=1072.937,205.997,419.745,173.867,27.178,154.838
C09069=1072.930,205.748,419.769,173.865,27.175,154.837
C09070=1072.925,205.499,419.793,173.862,27.172,154.837
C09071=1072.920,205.251,419.817,173.861,27.169,154.836
C09072=1072.914,205.002,419.841,173.858,27.166,154.836
C09073=1072.908,204.753,419.866,173.856,27.163,154.836
C09074=1072.903,204.504,419.889,173.854,27.160,154.835
C09075=1072.897,204.255,419.914,173.851,27.157,154.835
C09076=1072.891,204.006,419.938,173.850,27.154,154.834
C09077=1072.885,203.758,419.962,173.847,27.151,154.834
C09078=1072.880,203.509,419.986,173.845,27.148,154.834
C09079=1072.875,203.261,420.010,173.842,27.145,154.833
C09080=1072.868,203.012,420.034,173.840,27.142,154.833
C09081=1072.863,202.762,420.058,173.839,27.139,154.832
C09082=1072.858,202.514,420.082,173.836,27.136,154.832
C09083=1072.852,202.266,420.106,173.834,27.133,154.832
C09084=1072.846,202.016,420.130,173.831,27.130,154.831
C09085=1072.840,201.767,420.153,173.830,27.128,154.831
C09086=1072.835,201.519,420.178,173.827,27.125,154.831
C09087=1072.828,201.270,420.202,173.825,27.122,154.830
C09088=1072.823,201.021,420.226,173.822,27.119,154.830
C09089=1072.817,200.772,420.249,173.820,27.116,154.830
C09090=1072.811,200.524,420.273,173.819,27.114,154.829
C09091=1072.805,200.275,420.297,173.816,27.110,154.829
C09092=1072.800,200.026,420.320,173.814,27.107,154.828
C09093=1072.794,199.777,420.344,173.811,27.104,154.828
C09094=1072.788,199.529,420.368,173.810,27.102,154.828
C09095=1072.783,199.279,420.392,173.807,27.099,154.827
C09096=1072.777,199.031,420.416,173.805,27.096,154.827
C09097=1072.771,198.783,420.439,173.802,27.093,154.827
C09098=1072.766,198.533,420.463,173.801,27.090,154.826
C09099=1072.759,198.284,420.487,173.799,27.087,154.826
C09100=1072.754,198.035,420.510,173.796,27.085,154.826
C09101=1072.748,197.787,420.534,173.794,27.082,154.825
C09102=1072.743,197.538,420.558,173.792,27.079,154.825
C09103=1072.737,197.289,420.581,173.790,27.076,154.824
C09104=1072.730,197.040,420.605,173.787,27.073,154.824
C09105=1072.725,196.791,420.629,173.785,27.070,154.824
C09106=1072.719,196.543,420.652,173.783,27.068,154.823
